// TIA Portal project "Snake" (V16)

(* hardware
DEVICE "S71500/ET200MP station_1"  S7-1500 station
   slot 0: "Telaio di montaggio_0"  Rack  6ES7 590-1***0-0AA0
   slot 1: "PLC_1"  CPU 1515-2 PN  6ES7 515-2AM02-0AB0  V2.8
      slot 3: "Display CPU_1"  6ES7591-1BA00-0AA0
      slot 32768: "Interfaccia PROFINET_1"  X1
         slot 32769: "Porta_1"  X1 P1
         slot 32770: "Porta_2"  X1 P2
      slot 33024: "Interfaccia PROFINET_2"  X2
         slot 33025: "Porta_1"  X2 P1
      slot 34817: "Virtual CP interface port_1"  Virtual CP interface port  Virtual CP interface port
DEVICE "HMI_1"  TP2200 Comfort
   slot 0: "HMI_1"  TP2200 Comfort  6AV2 124-0XC02-0AX1  16.0.0.0
   slot 1: "HMI_RT_2"  TP2200 Comfort  6AV2 124-0XC02-0AX1  16.0.0.0
   slot 5: "HMI_1.IE_CP_1"  PROFINET Interface  16.0.0.0
      slot 1: "Interfaccia_1 PROFINET"  PROFINET Interface
         slot 1: "Porta_1"  Port
         slot 2: "Porta_2"  Port
   slot 6: "HMI_1.IE_CP_2"  PROFINET Interface  16.0.0.0
      slot 1: "PROFINET Interface_GBit"  PROFINET Interface
         slot 1: "Porta_1"  Port
   slot 7: "HMI_1.MPI/DP_CP_1"  MPI/DP Interface  16.0.0.0
*)

// ===== PLC "PLC_1"  CPU 1515-2 PN =====

VAR_GLOBAL CONSTANT   // PLC tag table "Constants"
   "SNAKE_START_NUM" : DInt := 3;
   "DIRECTION_UP" : Int := 1;
   "DIRECTION_DOWN" : Int := 2;
   "DIRECTION_RIGHT" : Int := 3;
   "DIRECTION_LEFT" : Int := 4;
   "FIELD_HEIGHT" : DInt := 10;
   "FIELD_LENGTH" : DInt := 20;
   "DIRECTION_NONE" : Int := 0;
   "POINTS_BASE" : UDInt := 50;
END_VAR

TYPE "st_FieldBlock"
   STRUCT
      SnakePresence : Bool;   // Snake block present
      ApplePresence : Bool;   // Apple block present
      Shifted : Bool;   // Block already shifted
      PreviousDirection : Int;   // Previous block direction (1 = Up, 2 = Down, 3 = Right, 4 = Left)
      HMI_Visualization : USInt;   // HMI visualization (0 = nothing / 1 = snake / 2 = apple)
   END_STRUCT;
END_TYPE

DATA_BLOCK "DB_Field"   // DB1
{ S7_Optimized_Access := 'TRUE' }
VERSION : 0.1
   VAR RETAIN
      Field : Array[1.."FIELD_HEIGHT", 1.."FIELD_LENGTH"] of "st_FieldBlock";
   END_VAR
BEGIN
END_DATA_BLOCK

DATA_BLOCK "DB_Commands"   // DB2
{ S7_Optimized_Access := 'TRUE' }
VERSION : 0.1
   VAR
      Cmd : Struct
         Start : Bool;   // Start command
         Stop : Bool;   // Stop command
         Pause : Bool;   // Pause command
         SnakeUp : Bool;
         SnakeDown : Bool;
         SnakeRight : Bool;
         SnakeLeft : Bool;
         Speed : Real;   // Speed (blocks per second)
      END_STRUCT;
      Sts : Struct
         GameActive : Bool;   // Game active
         PauseActive : Bool;   // Pause active
         SnakeLength : UDInt;
      END_STRUCT;
   END_VAR
   VAR RETAIN
      Points : Struct
         Actual : UDInt;
         LastGame : UDInt;
         BestGame : UDInt;
         BestLength : UDInt;
      END_STRUCT;
   END_VAR
BEGIN
END_DATA_BLOCK

DATA_BLOCK "FB_MainLogic_DB"   // DB3
{ S7_Optimized_Access := 'TRUE' }
VERSION : 0.1
// stored: InstanceOfName FB_MainLogic
"FB_MainLogic"
BEGIN
END_DATA_BLOCK

FUNCTION_BLOCK "FB_MainLogic"   // FB1, SCL
{ S7_Optimized_Access := 'TRUE' }
VERSION : 0.1
   VAR
      TON_Speed : TON_TIME;   // Timer used for game speed
      ResetTimer : Bool;
      Fp_GameStart : R_TRIG;   // Edge detection for game start
      Fn_GameStart : F_TRIG;
      SnakeHeadHeightIndex : DInt;   // Height index for snake head (used for starting the calculation loops for the movement)
      SnakeHeadLengthIndex : DInt;   // Length index for snake head (used for starting the calculation loops for the movement)
      PreviousDirection : Int;
      SnakeDirection : Int;   // Snake Direction
   END_VAR
   VAR_TEMP
      PointsToAdd : UDInt;
      IndexHeight : DInt;
      IndexLength : DInt;
      RandomAppleHeight : DInt;   // Random height index where to generate the apple
      RandomAppleLength : DInt;   // Random length index where to generate the apple
      CollisionWithSnake : Bool;
      CollisionWithWall : Bool;
      GenerateApple : Bool;
      ShiftFlag : Bool;   // Variable for snake movement
      LengthIndexToCheck : DInt;
      HeightIndexToCheck : DInt;
      CheckSnakeLength : UDInt;
      DirectionToCheck : Int;
   END_VAR
BEGIN

   REGION Game commands

       REGION Game start

           IF "DB_Commands".Cmd.Start AND NOT "DB_Commands".Sts.GameActive THEN
               IF "DB_Commands".Cmd.Speed > 0.0 THEN
                   "DB_Commands".Sts.GameActive := TRUE;
                   "DB_Commands".Sts.PauseActive := FALSE;
               END_IF;
               "DB_Commands".Cmd.Start := FALSE;
           ELSIF "DB_Commands".Sts.GameActive THEN
               "DB_Commands".Cmd.Start := FALSE;
           END_IF;

       END_REGION

       REGION Game stop

           IF "DB_Commands".Cmd.Stop OR ("DB_Commands".Cmd.Speed <= 0.0) THEN
               "DB_Commands".Sts.GameActive := FALSE;
               "DB_Commands".Sts.PauseActive := FALSE;
               "DB_Commands".Cmd.Stop := FALSE;
               "DB_Commands".Cmd.Start := FALSE;
           END_IF;

       END_REGION

       REGION Game Pause

           IF "DB_Commands".Cmd.Pause THEN
               IF "DB_Commands".Sts.GameActive THEN
                   "DB_Commands".Sts.PauseActive := NOT "DB_Commands".Sts.PauseActive;
               ELSE
                   "DB_Commands".Sts.PauseActive := FALSE;
               END_IF;
               "DB_Commands".Cmd.Pause := FALSE;
           END_IF;

       END_REGION

       REGION Game speed

           IF "DB_Commands".Cmd.Speed > 0.0 THEN

               #TON_Speed(IN := "DB_Commands".Sts.GameActive AND NOT "DB_Commands".Sts.PauseActive AND NOT #ResetTimer,
                          PT := REAL_TO_DINT((1.0 / "DB_Commands".Cmd.Speed) * 1000.0));

               #ResetTimer := #TON_Speed.Q;
               #ShiftFlag := #TON_Speed.Q;

           END_IF;

       END_REGION

       REGION Game points

           #PointsToAdd := REAL_TO_UDINT("DB_Commands".Cmd.Speed * UDINT_TO_REAL("POINTS_BASE"));

       END_REGION

       REGION Snake movements

           IF "DB_Commands".Sts.GameActive AND NOT "DB_Commands".Sts.PauseActive THEN

               IF #ShiftFlag THEN

                   //Up
                   IF "DB_Commands".Cmd.SnakeUp THEN
                       IF #SnakeDirection <> "DIRECTION_DOWN" THEN
                           #SnakeDirection := "DIRECTION_UP";
                       END_IF;
                       "DB_Commands".Cmd.SnakeUp := FALSE;
                       //Down
                   ELSIF "DB_Commands".Cmd.SnakeDown THEN
                       IF #SnakeDirection <> "DIRECTION_UP" THEN
                           #SnakeDirection := "DIRECTION_DOWN";
                       END_IF;
                       "DB_Commands".Cmd.SnakeDown := FALSE;
                       //Left
                   ELSIF "DB_Commands".Cmd.SnakeLeft THEN
                       IF #SnakeDirection <> "DIRECTION_RIGHT" THEN
                           #SnakeDirection := "DIRECTION_LEFT";
                       END_IF;
                       "DB_Commands".Cmd.SnakeLeft := FALSE;
                       //Right
                   ELSIF "DB_Commands".Cmd.SnakeRight THEN
                       IF #SnakeDirection <> "DIRECTION_LEFT" THEN
                           #SnakeDirection := "DIRECTION_RIGHT";
                       END_IF;
                       "DB_Commands".Cmd.SnakeRight := FALSE;
                   END_IF;

               END_IF;

           ELSE
               "DB_Commands".Cmd.SnakeUp := FALSE;
               "DB_Commands".Cmd.SnakeDown := FALSE;
               "DB_Commands".Cmd.SnakeLeft := FALSE;
               "DB_Commands".Cmd.SnakeRight := FALSE;
           END_IF;

       END_REGION

   END_REGION


   REGION Game logic

       REGION Check start and snake + apple creation

           #Fp_GameStart(CLK := "DB_Commands".Sts.GameActive);

           IF #Fp_GameStart.Q THEN

               //Reset actual points
               "DB_Commands".Points.Actual := 0;

               //Reset previous game
               FOR #IndexHeight := 1 TO "FIELD_HEIGHT" DO
                   FOR #IndexLength := 1 TO "FIELD_LENGTH" DO
                       "DB_Field".Field[#IndexHeight, #IndexLength].SnakePresence := FALSE;
                       "DB_Field".Field[#IndexHeight, #IndexLength].ApplePresence := FALSE;
                       "DB_Field".Field[#IndexHeight, #IndexLength].PreviousDirection := "DIRECTION_NONE";
                       "DB_Field".Field[#IndexHeight, #IndexLength].Shifted := FALSE;
                   END_FOR;
               END_FOR;

               //Check for starting indexes
               #SnakeHeadHeightIndex := "FIELD_HEIGHT" / 2; //5
               #SnakeHeadLengthIndex := "FIELD_LENGTH" / 2; //10

               //Set right direction for starting
               #SnakeDirection := #PreviousDirection := "DIRECTION_RIGHT";

               FOR #IndexLength := #SnakeHeadLengthIndex TO (#SnakeHeadLengthIndex - "SNAKE_START_NUM" + 1) BY -1 DO
                   "DB_Field".Field[#SnakeHeadHeightIndex, #IndexLength].SnakePresence := TRUE;
                   "DB_Field".Field[#SnakeHeadHeightIndex, #IndexLength].PreviousDirection := #SnakeDirection;
                   //Check for index bound
                   IF #IndexLength <= 1 THEN
                       EXIT;
                   END_IF;
               END_FOR;

               REGION Random number generation for apple

                   //Generate random number for apple creation
                   #RandomAppleHeight := "FC_RandomGen"(LowerLimit := 1, UpperLimit := "FIELD_HEIGHT");
                   #RandomAppleLength := "FC_RandomGen"(LowerLimit := 1, UpperLimit := "FIELD_LENGTH");

                   //Check if the numbers set are not already a snake block
                   WHILE "DB_Field".Field[#RandomAppleHeight, #RandomAppleLength].SnakePresence DO
                       //First time checking
                       IF NOT "DB_Field".Field[#RandomAppleHeight, #RandomAppleLength].SnakePresence THEN
                           EXIT;
                       END_IF;

                       //If there's the snake then change indexes
                       #RandomAppleHeight := #RandomAppleHeight + "FC_RandomGen"(LowerLimit := 1, UpperLimit := "FIELD_HEIGHT");
                       #RandomAppleHeight := #RandomAppleHeight MOD "FIELD_HEIGHT";
                       #RandomAppleLength := #RandomAppleLength + "FC_RandomGen"(LowerLimit := 1, UpperLimit := "FIELD_LENGTH");
                       #RandomAppleLength := #RandomAppleLength MOD "FIELD_LENGTH";

                   END_WHILE;

                   //Set apple presence
                   "DB_Field".Field[#RandomAppleHeight, #RandomAppleLength].ApplePresence := TRUE;

               END_REGION

           END_IF;

       END_REGION

       REGION Snake movement

           IF #ShiftFlag THEN

               //Reset collisions & vars
               #CollisionWithSnake := FALSE;
               #CollisionWithWall := FALSE;
               #GenerateApple := FALSE;

               //Reset Shifted vars
               FOR #IndexHeight := 1 TO "FIELD_HEIGHT" DO
                   FOR #IndexLength := 1 TO "FIELD_LENGTH" DO
                       "DB_Field".Field[#IndexHeight, #IndexLength].Shifted := FALSE;
                   END_FOR;
               END_FOR;

               //Check snake movement
               IF #SnakeDirection = "DIRECTION_RIGHT" THEN

                   REGION Right direction

                       //Check wall collision
                       IF (#SnakeHeadLengthIndex + 1) > "FIELD_LENGTH" THEN
                           #CollisionWithWall := TRUE;
                           "DB_Commands".Sts.GameActive := FALSE;
                       ELSE
                           //Check collision with other snake parts
                           IF "DB_Field".Field[#SnakeHeadHeightIndex, #SnakeHeadLengthIndex + 1].SnakePresence THEN
                               #CollisionWithSnake := TRUE;
                               "DB_Commands".Sts.GameActive := FALSE;
                           END_IF;
                       END_IF;

                       //Move if we have no collisions
                       IF NOT #CollisionWithWall AND NOT #CollisionWithSnake THEN
                           //Right direction starting with the head
                           //Shift snake head
                           "DB_Field".Field[#SnakeHeadHeightIndex, #SnakeHeadLengthIndex + 1].SnakePresence := "DB_Field".Field[#SnakeHeadHeightIndex, #SnakeHeadLengthIndex].SnakePresence;
                           "DB_Field".Field[#SnakeHeadHeightIndex, #SnakeHeadLengthIndex + 1].Shifted := TRUE;
                           "DB_Field".Field[#SnakeHeadHeightIndex, #SnakeHeadLengthIndex + 1].PreviousDirection := #PreviousDirection := "DIRECTION_RIGHT";
                           //If apple presence in the block then don't delete the snake presence to create the new block
                           IF "DB_Field".Field[#SnakeHeadHeightIndex, #SnakeHeadLengthIndex + 1].ApplePresence THEN
                               "DB_Field".Field[#SnakeHeadHeightIndex, #SnakeHeadLengthIndex + 1].ApplePresence := FALSE;
                               "DB_Field".Field[#SnakeHeadHeightIndex, #SnakeHeadLengthIndex].Shifted := TRUE;
                               "DB_Field".Field[#SnakeHeadHeightIndex, #SnakeHeadLengthIndex].PreviousDirection := "DIRECTION_RIGHT";
                               #GenerateApple := TRUE;
                           ELSE
                               "DB_Field".Field[#SnakeHeadHeightIndex, #SnakeHeadLengthIndex].SnakePresence := FALSE;
                               "DB_Field".Field[#SnakeHeadHeightIndex, #SnakeHeadLengthIndex].PreviousDirection := "DIRECTION_NONE";
                           END_IF;
                           //Set the new direction to check for snake movement
                           #DirectionToCheck := "DIRECTION_LEFT";
                           #LengthIndexToCheck := #SnakeHeadLengthIndex;
                           #HeightIndexToCheck := #SnakeHeadHeightIndex;
                           //And update the new snake head indexes
                           #SnakeHeadLengthIndex := #SnakeHeadLengthIndex + 1;

                       END_IF;

                   END_REGION

               ELSIF #SnakeDirection = "DIRECTION_LEFT" THEN

                   REGION Left direction

                       //Check wall collision
                       IF (#SnakeHeadLengthIndex - 1) < 1 THEN
                           #CollisionWithWall := TRUE;
                           "DB_Commands".Sts.GameActive := FALSE;
                       ELSE
                           //Check collision with other snake parts
                           IF "DB_Field".Field[#SnakeHeadHeightIndex, #SnakeHeadLengthIndex - 1].SnakePresence THEN
                               #CollisionWithSnake := TRUE;
                               "DB_Commands".Sts.GameActive := FALSE;
                           END_IF;
                       END_IF;

                       //Move if we have no collisions
                       IF NOT #CollisionWithWall AND NOT #CollisionWithSnake THEN
                           //Right direction starting with the head
                           //Shift snake head
                           "DB_Field".Field[#SnakeHeadHeightIndex, #SnakeHeadLengthIndex - 1].SnakePresence := "DB_Field".Field[#SnakeHeadHeightIndex, #SnakeHeadLengthIndex].SnakePresence;
                           "DB_Field".Field[#SnakeHeadHeightIndex, #SnakeHeadLengthIndex - 1].Shifted := TRUE;
                           "DB_Field".Field[#SnakeHeadHeightIndex, #SnakeHeadLengthIndex - 1].PreviousDirection := #PreviousDirection := "DIRECTION_LEFT";
                           //If apple presence in the block then don't delete the snake presence to create the new block
                           IF "DB_Field".Field[#SnakeHeadHeightIndex, #SnakeHeadLengthIndex - 1].ApplePresence THEN
                               "DB_Field".Field[#SnakeHeadHeightIndex, #SnakeHeadLengthIndex - 1].ApplePresence := FALSE;
                               "DB_Field".Field[#SnakeHeadHeightIndex, #SnakeHeadLengthIndex].Shifted := TRUE;
                               "DB_Field".Field[#SnakeHeadHeightIndex, #SnakeHeadLengthIndex].PreviousDirection := "DIRECTION_LEFT";
                               #GenerateApple := TRUE;
                           ELSE
                               "DB_Field".Field[#SnakeHeadHeightIndex, #SnakeHeadLengthIndex].SnakePresence := FALSE;
                               "DB_Field".Field[#SnakeHeadHeightIndex, #SnakeHeadLengthIndex].PreviousDirection := "DIRECTION_NONE";
                           END_IF;
                           //Set the new direction to check for snake movement
                           #DirectionToCheck := "DIRECTION_RIGHT";
                           #LengthIndexToCheck := #SnakeHeadLengthIndex;
                           #HeightIndexToCheck := #SnakeHeadHeightIndex;
                           //And update the new snake head indexes
                           #SnakeHeadLengthIndex := #SnakeHeadLengthIndex - 1;

                       END_IF;

                   END_REGION

               ELSIF #SnakeDirection = "DIRECTION_UP" THEN

                   REGION Up direction

                       //Check wall collision
                       IF (#SnakeHeadHeightIndex + 1) > "FIELD_HEIGHT" THEN
                           #CollisionWithWall := TRUE;
                           "DB_Commands".Sts.GameActive := FALSE;
                       ELSE
                           //Check collision with other snake parts
                           IF "DB_Field".Field[#SnakeHeadHeightIndex + 1, #SnakeHeadLengthIndex].SnakePresence THEN
                               #CollisionWithSnake := TRUE;
                               "DB_Commands".Sts.GameActive := FALSE;
                           END_IF;
                       END_IF;

                       //Move if we have no collisions
                       IF NOT #CollisionWithWall AND NOT #CollisionWithSnake THEN
                           //Right direction starting with the head
                           //Shift snake head
                           "DB_Field".Field[#SnakeHeadHeightIndex + 1, #SnakeHeadLengthIndex].SnakePresence := "DB_Field".Field[#SnakeHeadHeightIndex, #SnakeHeadLengthIndex].SnakePresence;
                           "DB_Field".Field[#SnakeHeadHeightIndex + 1, #SnakeHeadLengthIndex].Shifted := TRUE;
                           "DB_Field".Field[#SnakeHeadHeightIndex + 1, #SnakeHeadLengthIndex].PreviousDirection := #PreviousDirection := "DIRECTION_UP";
                           //If apple presence in the block then don't delete the snake presence to create the new block
                           IF "DB_Field".Field[#SnakeHeadHeightIndex + 1, #SnakeHeadLengthIndex].ApplePresence THEN
                               "DB_Field".Field[#SnakeHeadHeightIndex + 1, #SnakeHeadLengthIndex].ApplePresence := FALSE;
                               "DB_Field".Field[#SnakeHeadHeightIndex, #SnakeHeadLengthIndex].Shifted := TRUE;
                               "DB_Field".Field[#SnakeHeadHeightIndex, #SnakeHeadLengthIndex].PreviousDirection := "DIRECTION_UP";
                               #GenerateApple := TRUE;
                           ELSE
                               "DB_Field".Field[#SnakeHeadHeightIndex, #SnakeHeadLengthIndex].SnakePresence := FALSE;
                               "DB_Field".Field[#SnakeHeadHeightIndex, #SnakeHeadLengthIndex].PreviousDirection := "DIRECTION_NONE";
                           END_IF;
                           //Set the new direction to check for snake movement
                           #DirectionToCheck := "DIRECTION_DOWN";
                           #LengthIndexToCheck := #SnakeHeadLengthIndex;
                           #HeightIndexToCheck := #SnakeHeadHeightIndex;
                           //And update the new snake head indexes
                           #SnakeHeadHeightIndex := #SnakeHeadHeightIndex + 1;

                       END_IF;

                   END_REGION

               ELSIF #SnakeDirection = "DIRECTION_DOWN" THEN

                   REGION Down direction

                       //Check wall collision
                       IF (#SnakeHeadHeightIndex - 1) < 1 THEN
                           #CollisionWithWall := TRUE;
                           "DB_Commands".Sts.GameActive := FALSE;
                       ELSE
                           //Check collision with other snake parts
                           IF "DB_Field".Field[#SnakeHeadHeightIndex - 1, #SnakeHeadLengthIndex].SnakePresence THEN
                               #CollisionWithSnake := TRUE;
                               "DB_Commands".Sts.GameActive := FALSE;
                           END_IF;
                       END_IF;

                       //Move if we have no collisions
                       IF NOT #CollisionWithWall AND NOT #CollisionWithSnake THEN
                           //Right direction starting with the head
                           //Shift snake head
                           "DB_Field".Field[#SnakeHeadHeightIndex - 1, #SnakeHeadLengthIndex].SnakePresence := "DB_Field".Field[#SnakeHeadHeightIndex, #SnakeHeadLengthIndex].SnakePresence;
                           "DB_Field".Field[#SnakeHeadHeightIndex - 1, #SnakeHeadLengthIndex].Shifted := TRUE;
                           "DB_Field".Field[#SnakeHeadHeightIndex - 1, #SnakeHeadLengthIndex].PreviousDirection := #PreviousDirection := "DIRECTION_DOWN";
                           //If apple presence in the block then don't delete the snake presence to create the new block
                           IF "DB_Field".Field[#SnakeHeadHeightIndex - 1, #SnakeHeadLengthIndex].ApplePresence THEN
                               "DB_Field".Field[#SnakeHeadHeightIndex - 1, #SnakeHeadLengthIndex].ApplePresence := FALSE;
                               "DB_Field".Field[#SnakeHeadHeightIndex, #SnakeHeadLengthIndex].Shifted := TRUE;
                               "DB_Field".Field[#SnakeHeadHeightIndex, #SnakeHeadLengthIndex].PreviousDirection := "DIRECTION_DOWN";
                               #GenerateApple := TRUE;
                           ELSE
                               "DB_Field".Field[#SnakeHeadHeightIndex, #SnakeHeadLengthIndex].SnakePresence := FALSE;
                               "DB_Field".Field[#SnakeHeadHeightIndex, #SnakeHeadLengthIndex].PreviousDirection := "DIRECTION_NONE";
                           END_IF;
                           //Set the new direction to check for snake movement
                           #DirectionToCheck := "DIRECTION_UP";
                           #LengthIndexToCheck := #SnakeHeadLengthIndex;
                           #HeightIndexToCheck := #SnakeHeadHeightIndex;
                           //And update the new snake head indexes
                           #SnakeHeadHeightIndex := #SnakeHeadHeightIndex - 1;

                       END_IF;

                   END_REGION

               END_IF;

               REGION Snake shifts

                   IF NOT #CollisionWithWall AND NOT #CollisionWithSnake AND NOT #GenerateApple THEN

                       WHILE #DirectionToCheck <> "DIRECTION_NONE" DO

                           //Check the left direction
                           IF #DirectionToCheck = "DIRECTION_LEFT" THEN
                               FOR #IndexLength := (#LengthIndexToCheck - 1) TO 1 BY -1 DO
                                   IF "DB_Field".Field[#HeightIndexToCheck, #IndexLength].SnakePresence AND
                                       NOT "DB_Field".Field[#HeightIndexToCheck, #IndexLength].Shifted AND
                                       "DB_Field".Field[#HeightIndexToCheck, #IndexLength].PreviousDirection <> "DIRECTION_LEFT" THEN

                                       "DB_Field".Field[#HeightIndexToCheck, #IndexLength + 1].SnakePresence := "DB_Field".Field[#HeightIndexToCheck, #IndexLength].SnakePresence;
                                       "DB_Field".Field[#HeightIndexToCheck, #IndexLength + 1].PreviousDirection := #PreviousDirection;
                                       "DB_Field".Field[#HeightIndexToCheck, #IndexLength + 1].Shifted := TRUE;

                                       "DB_Field".Field[#HeightIndexToCheck, #IndexLength].SnakePresence := FALSE;
                                       "DB_Field".Field[#HeightIndexToCheck, #IndexLength].PreviousDirection := "DIRECTION_NONE";
                                       #LengthIndexToCheck := #IndexLength;
                                   ELSE
                                       EXIT;
                                   END_IF;
                               END_FOR;
                               //When the shift is finished check the other directions
                               #DirectionToCheck := "DIRECTION_NONE";
                               //Check up
                               IF (#HeightIndexToCheck + 1) <= "FIELD_HEIGHT" THEN
                                   IF "DB_Field".Field[#HeightIndexToCheck + 1, #LengthIndexToCheck].SnakePresence AND
                                       NOT "DB_Field".Field[#HeightIndexToCheck + 1, #LengthIndexToCheck].Shifted THEN
                                       #DirectionToCheck := "DIRECTION_UP";
                                       #PreviousDirection := "DIRECTION_DOWN";
                                   END_IF;
                               END_IF;
                               //Check down
                               IF (#HeightIndexToCheck - 1) >= 1 THEN
                                   IF "DB_Field".Field[#HeightIndexToCheck - 1, #LengthIndexToCheck].SnakePresence AND
                                       NOT "DB_Field".Field[#HeightIndexToCheck - 1, #LengthIndexToCheck].Shifted THEN
                                       #DirectionToCheck := "DIRECTION_DOWN";
                                       #PreviousDirection := "DIRECTION_UP";
                                   END_IF;
                               END_IF;

                               //Check the right direction
                           ELSIF #DirectionToCheck = "DIRECTION_RIGHT" THEN
                               FOR #IndexLength := (#LengthIndexToCheck + 1) TO "FIELD_LENGTH" DO
                                   IF "DB_Field".Field[#HeightIndexToCheck, #IndexLength].SnakePresence AND
                                       NOT "DB_Field".Field[#HeightIndexToCheck, #IndexLength].Shifted AND
                                       "DB_Field".Field[#HeightIndexToCheck, #IndexLength].PreviousDirection <> "DIRECTION_RIGHT" THEN

                                       "DB_Field".Field[#HeightIndexToCheck, #IndexLength - 1].SnakePresence := "DB_Field".Field[#HeightIndexToCheck, #IndexLength].SnakePresence;
                                       "DB_Field".Field[#HeightIndexToCheck, #IndexLength - 1].PreviousDirection := #PreviousDirection;
                                       "DB_Field".Field[#HeightIndexToCheck, #IndexLength - 1].Shifted := TRUE;

                                       "DB_Field".Field[#HeightIndexToCheck, #IndexLength].SnakePresence := FALSE;
                                       "DB_Field".Field[#HeightIndexToCheck, #IndexLength].PreviousDirection := "DIRECTION_NONE";
                                       #LengthIndexToCheck := #IndexLength;
                                   ELSE
                                       EXIT;
                                   END_IF;
                               END_FOR;
                               //When the shift is finished check the other directions
                               #DirectionToCheck := "DIRECTION_NONE";
                               //Check up
                               IF (#HeightIndexToCheck + 1) <= "FIELD_HEIGHT" THEN
                                   IF "DB_Field".Field[#HeightIndexToCheck + 1, #LengthIndexToCheck].SnakePresence AND
                                       NOT "DB_Field".Field[#HeightIndexToCheck + 1, #LengthIndexToCheck].Shifted THEN
                                       #DirectionToCheck := "DIRECTION_UP";
                                       #PreviousDirection := "DIRECTION_DOWN";
                                   END_IF;
                               END_IF;
                               //Check down
                               IF (#HeightIndexToCheck - 1) >= 1 THEN
                                   IF "DB_Field".Field[#HeightIndexToCheck - 1, #LengthIndexToCheck].SnakePresence AND
                                       NOT "DB_Field".Field[#HeightIndexToCheck - 1, #LengthIndexToCheck].Shifted THEN
                                       #DirectionToCheck := "DIRECTION_DOWN";
                                       #PreviousDirection := "DIRECTION_UP";
                                   END_IF;
                               END_IF;

                               //Check the down direction
                           ELSIF #DirectionToCheck = "DIRECTION_DOWN" THEN
                               FOR #IndexHeight := (#HeightIndexToCheck - 1) TO 1 BY -1 DO
                                   IF "DB_Field".Field[#IndexHeight, #LengthIndexToCheck].SnakePresence AND
                                       NOT "DB_Field".Field[#IndexHeight, #LengthIndexToCheck].Shifted AND
                                       "DB_Field".Field[#IndexHeight, #LengthIndexToCheck].PreviousDirection <> "DIRECTION_DOWN" THEN

                                       "DB_Field".Field[#IndexHeight + 1, #LengthIndexToCheck].SnakePresence := "DB_Field".Field[#IndexHeight, #LengthIndexToCheck].SnakePresence;
                                       "DB_Field".Field[#IndexHeight + 1, #LengthIndexToCheck].PreviousDirection := #PreviousDirection;
                                       "DB_Field".Field[#IndexHeight + 1, #LengthIndexToCheck].Shifted := TRUE;

                                       "DB_Field".Field[#IndexHeight, #LengthIndexToCheck].SnakePresence := FALSE;
                                       "DB_Field".Field[#IndexHeight, #LengthIndexToCheck].PreviousDirection := "DIRECTION_NONE";
                                       #HeightIndexToCheck := #IndexHeight;
                                   ELSE
                                       EXIT;
                                   END_IF;
                               END_FOR;
                               //When the shift is finished check the other directions
                               #DirectionToCheck := "DIRECTION_NONE";
                               //Check left
                               IF (#LengthIndexToCheck - 1) >= 1 THEN
                                   IF "DB_Field".Field[#HeightIndexToCheck, #LengthIndexToCheck - 1].SnakePresence AND
                                       NOT "DB_Field".Field[#HeightIndexToCheck, #LengthIndexToCheck - 1].Shifted THEN
                                       #DirectionToCheck := "DIRECTION_LEFT";
                                       #PreviousDirection := "DIRECTION_RIGHT";
                                   END_IF;
                               END_IF;
                               //Check down
                               IF (#LengthIndexToCheck + 1) <= "FIELD_LENGTH" THEN
                                   IF "DB_Field".Field[#HeightIndexToCheck, #LengthIndexToCheck + 1].SnakePresence AND
                                       NOT "DB_Field".Field[#HeightIndexToCheck, #LengthIndexToCheck + 1].Shifted THEN
                                       #DirectionToCheck := "DIRECTION_RIGHT";
                                       #PreviousDirection := "DIRECTION_LEFT";
                                   END_IF;
                               END_IF;

                               //Check the up direction
                           ELSIF #DirectionToCheck = "DIRECTION_UP" THEN
                               FOR #IndexHeight := (#HeightIndexToCheck + 1) TO "FIELD_HEIGHT" DO
                                   IF "DB_Field".Field[#IndexHeight, #LengthIndexToCheck].SnakePresence AND
                                       NOT "DB_Field".Field[#IndexHeight, #LengthIndexToCheck].Shifted AND
                                       "DB_Field".Field[#IndexHeight, #LengthIndexToCheck].PreviousDirection <> "DIRECTION_UP" THEN

                                       "DB_Field".Field[#IndexHeight - 1, #LengthIndexToCheck].SnakePresence := "DB_Field".Field[#IndexHeight, #LengthIndexToCheck].SnakePresence;
                                       "DB_Field".Field[#IndexHeight - 1, #LengthIndexToCheck].PreviousDirection := #PreviousDirection;
                                       "DB_Field".Field[#IndexHeight - 1, #LengthIndexToCheck].Shifted := TRUE;

                                       "DB_Field".Field[#IndexHeight, #LengthIndexToCheck].SnakePresence := FALSE;
                                       "DB_Field".Field[#IndexHeight, #LengthIndexToCheck].PreviousDirection := "DIRECTION_NONE";
                                       #HeightIndexToCheck := #IndexHeight;
                                   ELSE
                                       EXIT;
                                   END_IF;
                               END_FOR;
                               //When the shift is finished check the other directions
                               #DirectionToCheck := "DIRECTION_NONE";
                               //Check left
                               IF (#LengthIndexToCheck - 1) >= 1 THEN
                                   IF "DB_Field".Field[#HeightIndexToCheck, #LengthIndexToCheck - 1].SnakePresence AND
                                       NOT "DB_Field".Field[#HeightIndexToCheck, #LengthIndexToCheck - 1].Shifted THEN
                                       #DirectionToCheck := "DIRECTION_LEFT";
                                       #PreviousDirection := "DIRECTION_RIGHT";
                                   END_IF;
                               END_IF;
                               //Check down
                               IF (#LengthIndexToCheck + 1) <= "FIELD_LENGTH" THEN
                                   IF "DB_Field".Field[#HeightIndexToCheck, #LengthIndexToCheck + 1].SnakePresence AND
                                       NOT "DB_Field".Field[#HeightIndexToCheck, #LengthIndexToCheck + 1].Shifted THEN
                                       #DirectionToCheck := "DIRECTION_RIGHT";
                                       #PreviousDirection := "DIRECTION_LEFT";
                                   END_IF;
                               END_IF;
                           END_IF;

                       END_WHILE;

                   END_IF;

               END_REGION

               REGION Check for new apple generation

                   IF #GenerateApple THEN

                       //Increase score
                       "DB_Commands".Points.Actual := "DB_Commands".Points.Actual + #PointsToAdd;

                       //Generate random number for apple creation
                       #RandomAppleHeight := "FC_RandomGen"(LowerLimit := 1, UpperLimit := "FIELD_HEIGHT");
                       #RandomAppleLength := "FC_RandomGen"(LowerLimit := 1, UpperLimit := "FIELD_LENGTH");

                       //Check if the numbers set are not already a snake block
                       WHILE "DB_Field".Field[#RandomAppleHeight, #RandomAppleLength].SnakePresence DO
                           //First time checking
                           IF NOT "DB_Field".Field[#RandomAppleHeight, #RandomAppleLength].SnakePresence THEN
                               EXIT;
                           END_IF;

                           //If there's the snake then change indexes
                           #RandomAppleHeight := #RandomAppleHeight + "FC_RandomGen"(LowerLimit := 1, UpperLimit := "FIELD_HEIGHT");
                           #RandomAppleHeight := #RandomAppleHeight MOD "FIELD_HEIGHT";
                           #RandomAppleLength := #RandomAppleLength + "FC_RandomGen"(LowerLimit := 1, UpperLimit := "FIELD_LENGTH");
                           #RandomAppleLength := #RandomAppleLength MOD "FIELD_LENGTH";

                       END_WHILE;

                       //Set apple presence
                       "DB_Field".Field[#RandomAppleHeight, #RandomAppleLength].ApplePresence := TRUE;

                   END_IF;

               END_REGION

           END_IF;

       END_REGION

       REGION Snake length calculation

           "DB_Commands".Sts.SnakeLength := 0;
           FOR #IndexHeight := 1 TO "FIELD_HEIGHT" DO
               FOR #IndexLength := 1 TO "FIELD_LENGTH" DO
                   IF "DB_Field".Field[#IndexHeight, #IndexLength].SnakePresence THEN
                       "DB_Commands".Sts.SnakeLength := "DB_Commands".Sts.SnakeLength + 1;
                   END_IF;
               END_FOR;
           END_FOR;

       END_REGION

       REGION Check for game end to score points

           #Fn_GameStart(CLK := "DB_Commands".Sts.GameActive);

           IF #Fn_GameStart.Q THEN
               "DB_Commands".Points.LastGame := "DB_Commands".Points.Actual;
               IF "DB_Commands".Points.LastGame > "DB_Commands".Points.BestGame THEN
                   "DB_Commands".Points.BestGame := "DB_Commands".Points.LastGame;
               END_IF;
               IF "DB_Commands".Sts.SnakeLength > "DB_Commands".Points.BestLength THEN
                   "DB_Commands".Points.BestLength := "DB_Commands".Sts.SnakeLength;
               END_IF;
           END_IF;

       END_REGION

   END_REGION
END_FUNCTION_BLOCK

FUNCTION "FC_RandomGen" : DInt   // FC1, LAD
{ S7_Optimized_Access := 'TRUE' }
VERSION : 0.1
   VAR_INPUT
      LowerLimit : DInt;
      UpperLimit : DInt;
   END_VAR
   VAR_TEMP
      DateTime : DTL;
      ReadTimeRetVal : Int;
      NanoSecMod : Int;
      ChoppedTime : Int;
      UShift : UInt;
      SemiRandom : UInt;
      NormalizedRandom : Real;
   END_VAR
BEGIN

REGION Network 1: Read actual date/time to retrieve nanoseconds
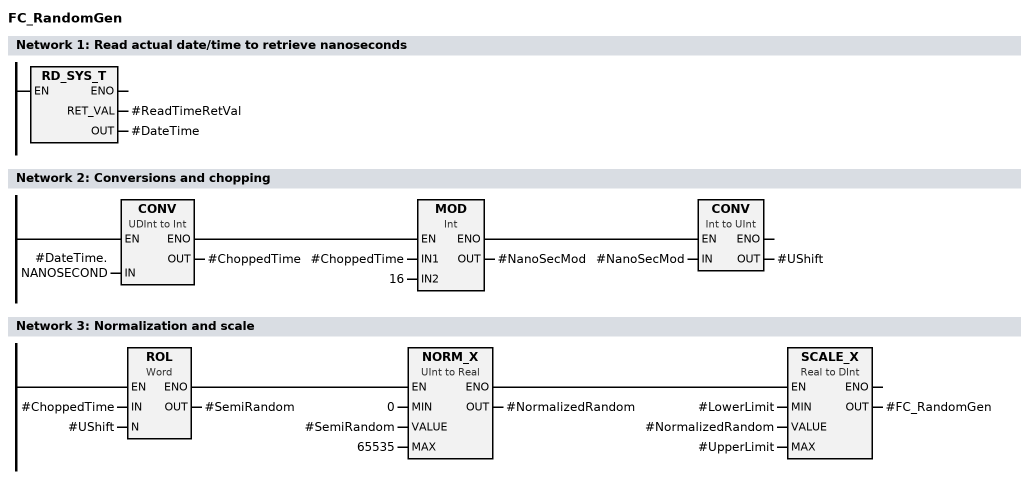
   #ReadTimeRetVal := RD_SYS_T(OUT => #DateTime);
END_REGION

REGION Network 2: Conversions and chopping
   RUNG wire#powerrail
      { S7_Templates := "[SrcType := UDInt, DestType := Int]" } Convert(in := #DateTime.NANOSECOND, out => #ChoppedTime)
      { S7_Templates := "SrcType := Int" } Mod(in1 := #ChoppedTime, in2 := 16, out => #NanoSecMod)
      { S7_Templates := "[SrcType := Int, DestType := UInt]" } Convert(in := #NanoSecMod, out => #UShift)
   END_RUNG
   // the same network as SCL:
   #ChoppedTime := UDINT_TO_INT(#DateTime.NANOSECOND);
   #NanoSecMod := #ChoppedTime MOD 16;
   #UShift := INT_TO_UINT(#NanoSecMod);
END_REGION

REGION Network 3: Normalization and scale
   #SemiRandom := ROL(IN := #ChoppedTime, N := #UShift);
   #NormalizedRandom := NORM_X(MIN := 0, VALUE := #SemiRandom, MAX := 65535);
   #FC_RandomGen := SCALE_X(MIN := #LowerLimit, VALUE := #NormalizedRandom, MAX := #UpperLimit);
END_REGION
END_FUNCTION

ORGANIZATION_BLOCK "Main"   // OB1, LAD, ProgramCycle
TITLE = "Main Program Sweep (Cycle)"
{ S7_Optimized_Access := 'TRUE' }
VERSION : 0.1
   VAR_INPUT
      Initial_Call : Bool;   // Initial call of this OB
      Remanence : Bool;   // =True, if remanent data are available
   END_VAR
   VAR_TEMP
      IndexHeight : DInt;
      IndexLength : DInt;
   END_VAR
BEGIN

REGION Network 1
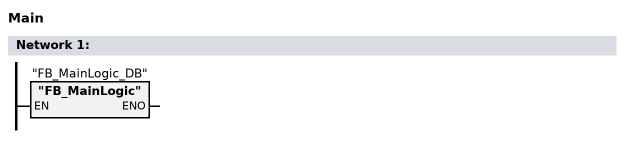
   RUNG wire#powerrail
      "FB_MainLogic_DB"()
   END_RUNG
   // the same network as SCL:
   "FB_MainLogic_DB"();   // "FB_MainLogic"
END_REGION

REGION Network 2 (SCL): Visualizzazione blocchi per HMI
   FOR #IndexHeight := 1 TO "FIELD_HEIGHT" DO
       FOR #IndexLength := 1 TO "FIELD_LENGTH" DO
           IF "DB_Field".Field[#IndexHeight, #IndexLength].SnakePresence THEN
               "DB_Field".Field[#IndexHeight, #IndexLength].HMI_Visualization := 1;
           ELSIF "DB_Field".Field[#IndexHeight, #IndexLength].ApplePresence THEN
               "DB_Field".Field[#IndexHeight, #IndexLength].HMI_Visualization := 2;
           ELSE
               "DB_Field".Field[#IndexHeight, #IndexLength].HMI_Visualization := 0;
           END_IF;
       END_FOR;
   END_FOR;
END_REGION
END_ORGANIZATION_BLOCK

(* ===== HMI "HMI_RT_2" =====
system functions are stored by id; their names below are inferred from use
connection "HMI_Collegamento_1": ETHERNET, S7_1500_OMS

HMI tags "Tabella delle variabili standard"
   "Variabile_Numero di pagina" : UInt, internal
   "DB_Field_Field{1,1}_HMI_Visualization" : USInt = PLC DB_Field.Field[1,1].HMI_Visualization AT %DB1.DBW0, 100 ms
   "DB_Field_Field{1,2}_HMI_Visualization" : USInt = PLC DB_Field.Field[1,2].HMI_Visualization AT %DB1.DBW0, 100 ms
   "DB_Field_Field{1,3}_HMI_Visualization" : USInt = PLC DB_Field.Field[1,3].HMI_Visualization AT %DB1.DBW0, 100 ms
   "DB_Field_Field{1,4}_HMI_Visualization" : USInt = PLC DB_Field.Field[1,4].HMI_Visualization AT %DB1.DBW0, 100 ms
   "DB_Field_Field{1,5}_HMI_Visualization" : USInt = PLC DB_Field.Field[1,5].HMI_Visualization AT %DB1.DBW0, 100 ms
   "DB_Field_Field{1,6}_HMI_Visualization" : USInt = PLC DB_Field.Field[1,6].HMI_Visualization AT %DB1.DBW0, 100 ms
   "DB_Field_Field{1,7}_HMI_Visualization" : USInt = PLC DB_Field.Field[1,7].HMI_Visualization AT %DB1.DBW0, 100 ms
   "DB_Field_Field{1,8}_HMI_Visualization" : USInt = PLC DB_Field.Field[1,8].HMI_Visualization AT %DB1.DBW0, 100 ms
   "DB_Field_Field{1,9}_HMI_Visualization" : USInt = PLC DB_Field.Field[1,9].HMI_Visualization AT %DB1.DBW0, 100 ms
   "DB_Field_Field{1,10}_HMI_Visualization" : USInt = PLC DB_Field.Field[1,10].HMI_Visualization AT %DB1.DBW0, 100 ms
   "DB_Field_Field{1,11}_HMI_Visualization" : USInt = PLC DB_Field.Field[1,11].HMI_Visualization AT %DB1.DBW0, 100 ms
   "DB_Field_Field{1,12}_HMI_Visualization" : USInt = PLC DB_Field.Field[1,12].HMI_Visualization AT %DB1.DBW0, 100 ms
   "DB_Field_Field{1,13}_HMI_Visualization" : USInt = PLC DB_Field.Field[1,13].HMI_Visualization AT %DB1.DBW0, 100 ms
   "DB_Field_Field{1,14}_HMI_Visualization" : USInt = PLC DB_Field.Field[1,14].HMI_Visualization AT %DB1.DBW0, 100 ms
   "DB_Field_Field{1,15}_HMI_Visualization" : USInt = PLC DB_Field.Field[1,15].HMI_Visualization AT %DB1.DBW0, 100 ms
   "DB_Field_Field{1,16}_HMI_Visualization" : USInt = PLC DB_Field.Field[1,16].HMI_Visualization AT %DB1.DBW0, 100 ms
   "DB_Field_Field{1,17}_HMI_Visualization" : USInt = PLC DB_Field.Field[1,17].HMI_Visualization AT %DB1.DBW0, 100 ms
   "DB_Field_Field{1,18}_HMI_Visualization" : USInt = PLC DB_Field.Field[1,18].HMI_Visualization AT %DB1.DBW0, 100 ms
   "DB_Field_Field{1,19}_HMI_Visualization" : USInt = PLC DB_Field.Field[1,19].HMI_Visualization AT %DB1.DBW0, 100 ms
   "DB_Field_Field{1,20}_HMI_Visualization" : USInt = PLC DB_Field.Field[1,20].HMI_Visualization AT %DB1.DBW0, 100 ms
   "DB_Field_Field{2,1}_HMI_Visualization" : USInt = PLC DB_Field.Field[2,1].HMI_Visualization AT %DB1.DBW0, 100 ms
   "DB_Field_Field{2,2}_HMI_Visualization" : USInt = PLC DB_Field.Field[2,2].HMI_Visualization AT %DB1.DBW0, 100 ms
   "DB_Field_Field{2,3}_HMI_Visualization" : USInt = PLC DB_Field.Field[2,3].HMI_Visualization AT %DB1.DBW0, 100 ms
   "DB_Field_Field{2,4}_HMI_Visualization" : USInt = PLC DB_Field.Field[2,4].HMI_Visualization AT %DB1.DBW0, 100 ms
   "DB_Field_Field{2,5}_HMI_Visualization" : USInt = PLC DB_Field.Field[2,5].HMI_Visualization AT %DB1.DBW0, 100 ms
   "DB_Field_Field{2,6}_HMI_Visualization" : USInt = PLC DB_Field.Field[2,6].HMI_Visualization AT %DB1.DBW0, 100 ms
   "DB_Field_Field{2,7}_HMI_Visualization" : USInt = PLC DB_Field.Field[2,7].HMI_Visualization AT %DB1.DBW0, 100 ms
   "DB_Field_Field{2,8}_HMI_Visualization" : USInt = PLC DB_Field.Field[2,8].HMI_Visualization AT %DB1.DBW0, 100 ms
   "DB_Field_Field{2,9}_HMI_Visualization" : USInt = PLC DB_Field.Field[2,9].HMI_Visualization AT %DB1.DBW0, 100 ms
   "DB_Field_Field{2,10}_HMI_Visualization" : USInt = PLC DB_Field.Field[2,10].HMI_Visualization AT %DB1.DBW0, 100 ms
   "DB_Field_Field{2,11}_HMI_Visualization" : USInt = PLC DB_Field.Field[2,11].HMI_Visualization AT %DB1.DBW0, 100 ms
   "DB_Field_Field{2,12}_HMI_Visualization" : USInt = PLC DB_Field.Field[2,12].HMI_Visualization AT %DB1.DBW0, 100 ms
   "DB_Field_Field{2,13}_HMI_Visualization" : USInt = PLC DB_Field.Field[2,13].HMI_Visualization AT %DB1.DBW0, 100 ms
   "DB_Field_Field{2,14}_HMI_Visualization" : USInt = PLC DB_Field.Field[2,14].HMI_Visualization AT %DB1.DBW0, 100 ms
   "DB_Field_Field{2,15}_HMI_Visualization" : USInt = PLC DB_Field.Field[2,15].HMI_Visualization AT %DB1.DBW0, 100 ms
   "DB_Field_Field{2,16}_HMI_Visualization" : USInt = PLC DB_Field.Field[2,16].HMI_Visualization AT %DB1.DBW0, 100 ms
   "DB_Field_Field{2,17}_HMI_Visualization" : USInt = PLC DB_Field.Field[2,17].HMI_Visualization AT %DB1.DBW0, 100 ms
   "DB_Field_Field{2,18}_HMI_Visualization" : USInt = PLC DB_Field.Field[2,18].HMI_Visualization AT %DB1.DBW0, 100 ms
   "DB_Field_Field{2,19}_HMI_Visualization" : USInt = PLC DB_Field.Field[2,19].HMI_Visualization AT %DB1.DBW0, 100 ms
   "DB_Field_Field{2,20}_HMI_Visualization" : USInt = PLC DB_Field.Field[2,20].HMI_Visualization AT %DB1.DBW0, 100 ms
   "DB_Field_Field{3,1}_HMI_Visualization" : USInt = PLC DB_Field.Field[3,1].HMI_Visualization AT %DB1.DBW0, 100 ms
   "DB_Field_Field{3,2}_HMI_Visualization" : USInt = PLC DB_Field.Field[3,2].HMI_Visualization AT %DB1.DBW0, 100 ms
   "DB_Field_Field{3,3}_HMI_Visualization" : USInt = PLC DB_Field.Field[3,3].HMI_Visualization AT %DB1.DBW0, 100 ms
   "DB_Field_Field{3,4}_HMI_Visualization" : USInt = PLC DB_Field.Field[3,4].HMI_Visualization AT %DB1.DBW0, 100 ms
   "DB_Field_Field{3,5}_HMI_Visualization" : USInt = PLC DB_Field.Field[3,5].HMI_Visualization AT %DB1.DBW0, 100 ms
   "DB_Field_Field{3,6}_HMI_Visualization" : USInt = PLC DB_Field.Field[3,6].HMI_Visualization AT %DB1.DBW0, 100 ms
   "DB_Field_Field{3,7}_HMI_Visualization" : USInt = PLC DB_Field.Field[3,7].HMI_Visualization AT %DB1.DBW0, 100 ms
   "DB_Field_Field{3,8}_HMI_Visualization" : USInt = PLC DB_Field.Field[3,8].HMI_Visualization AT %DB1.DBW0, 100 ms
   "DB_Field_Field{3,9}_HMI_Visualization" : USInt = PLC DB_Field.Field[3,9].HMI_Visualization AT %DB1.DBW0, 100 ms
   "DB_Field_Field{3,10}_HMI_Visualization" : USInt = PLC DB_Field.Field[3,10].HMI_Visualization AT %DB1.DBW0, 100 ms
   "DB_Field_Field{3,11}_HMI_Visualization" : USInt = PLC DB_Field.Field[3,11].HMI_Visualization AT %DB1.DBW0, 100 ms
   "DB_Field_Field{3,12}_HMI_Visualization" : USInt = PLC DB_Field.Field[3,12].HMI_Visualization AT %DB1.DBW0, 100 ms
   "DB_Field_Field{3,13}_HMI_Visualization" : USInt = PLC DB_Field.Field[3,13].HMI_Visualization AT %DB1.DBW0, 100 ms
   "DB_Field_Field{3,14}_HMI_Visualization" : USInt = PLC DB_Field.Field[3,14].HMI_Visualization AT %DB1.DBW0, 100 ms
   "DB_Field_Field{3,15}_HMI_Visualization" : USInt = PLC DB_Field.Field[3,15].HMI_Visualization AT %DB1.DBW0, 100 ms
   "DB_Field_Field{3,16}_HMI_Visualization" : USInt = PLC DB_Field.Field[3,16].HMI_Visualization AT %DB1.DBW0, 100 ms
   "DB_Field_Field{3,17}_HMI_Visualization" : USInt = PLC DB_Field.Field[3,17].HMI_Visualization AT %DB1.DBW0, 100 ms
   "DB_Field_Field{3,18}_HMI_Visualization" : USInt = PLC DB_Field.Field[3,18].HMI_Visualization AT %DB1.DBW0, 100 ms
   "DB_Field_Field{3,19}_HMI_Visualization" : USInt = PLC DB_Field.Field[3,19].HMI_Visualization AT %DB1.DBW0, 100 ms
   "DB_Field_Field{3,20}_HMI_Visualization" : USInt = PLC DB_Field.Field[3,20].HMI_Visualization AT %DB1.DBW0, 100 ms
   "DB_Field_Field{4,1}_HMI_Visualization" : USInt = PLC DB_Field.Field[4,1].HMI_Visualization AT %DB1.DBW0, 100 ms
   "DB_Field_Field{4,2}_HMI_Visualization" : USInt = PLC DB_Field.Field[4,2].HMI_Visualization AT %DB1.DBW0, 100 ms
   "DB_Field_Field{4,3}_HMI_Visualization" : USInt = PLC DB_Field.Field[4,3].HMI_Visualization AT %DB1.DBW0, 100 ms
   "DB_Field_Field{4,4}_HMI_Visualization" : USInt = PLC DB_Field.Field[4,4].HMI_Visualization AT %DB1.DBW0, 100 ms
   "DB_Field_Field{4,5}_HMI_Visualization" : USInt = PLC DB_Field.Field[4,5].HMI_Visualization AT %DB1.DBW0, 100 ms
   "DB_Field_Field{4,6}_HMI_Visualization" : USInt = PLC DB_Field.Field[4,6].HMI_Visualization AT %DB1.DBW0, 100 ms
   "DB_Field_Field{4,7}_HMI_Visualization" : USInt = PLC DB_Field.Field[4,7].HMI_Visualization AT %DB1.DBW0, 100 ms
   "DB_Field_Field{4,8}_HMI_Visualization" : USInt = PLC DB_Field.Field[4,8].HMI_Visualization AT %DB1.DBW0, 100 ms
   "DB_Field_Field{4,9}_HMI_Visualization" : USInt = PLC DB_Field.Field[4,9].HMI_Visualization AT %DB1.DBW0, 100 ms
   "DB_Field_Field{4,10}_HMI_Visualization" : USInt = PLC DB_Field.Field[4,10].HMI_Visualization AT %DB1.DBW0, 100 ms
   "DB_Field_Field{4,11}_HMI_Visualization" : USInt = PLC DB_Field.Field[4,11].HMI_Visualization AT %DB1.DBW0, 100 ms
   "DB_Field_Field{4,12}_HMI_Visualization" : USInt = PLC DB_Field.Field[4,12].HMI_Visualization AT %DB1.DBW0, 100 ms
   "DB_Field_Field{4,13}_HMI_Visualization" : USInt = PLC DB_Field.Field[4,13].HMI_Visualization AT %DB1.DBW0, 100 ms
   "DB_Field_Field{4,14}_HMI_Visualization" : USInt = PLC DB_Field.Field[4,14].HMI_Visualization AT %DB1.DBW0, 100 ms
   "DB_Field_Field{4,15}_HMI_Visualization" : USInt = PLC DB_Field.Field[4,15].HMI_Visualization AT %DB1.DBW0, 100 ms
   "DB_Field_Field{4,16}_HMI_Visualization" : USInt = PLC DB_Field.Field[4,16].HMI_Visualization AT %DB1.DBW0, 100 ms
   "DB_Field_Field{4,17}_HMI_Visualization" : USInt = PLC DB_Field.Field[4,17].HMI_Visualization AT %DB1.DBW0, 100 ms
   "DB_Field_Field{4,18}_HMI_Visualization" : USInt = PLC DB_Field.Field[4,18].HMI_Visualization AT %DB1.DBW0, 100 ms
   "DB_Field_Field{4,19}_HMI_Visualization" : USInt = PLC DB_Field.Field[4,19].HMI_Visualization AT %DB1.DBW0, 100 ms
   "DB_Field_Field{4,20}_HMI_Visualization" : USInt = PLC DB_Field.Field[4,20].HMI_Visualization AT %DB1.DBW0, 100 ms
   "DB_Field_Field{5,1}_HMI_Visualization" : USInt = PLC DB_Field.Field[5,1].HMI_Visualization AT %DB1.DBW0, 100 ms
   "DB_Field_Field{5,2}_HMI_Visualization" : USInt = PLC DB_Field.Field[5,2].HMI_Visualization AT %DB1.DBW0, 100 ms
   "DB_Field_Field{5,3}_HMI_Visualization" : USInt = PLC DB_Field.Field[5,3].HMI_Visualization AT %DB1.DBW0, 100 ms
   "DB_Field_Field{5,4}_HMI_Visualization" : USInt = PLC DB_Field.Field[5,4].HMI_Visualization AT %DB1.DBW0, 100 ms
   "DB_Field_Field{5,5}_HMI_Visualization" : USInt = PLC DB_Field.Field[5,5].HMI_Visualization AT %DB1.DBW0, 100 ms
   "DB_Field_Field{5,6}_HMI_Visualization" : USInt = PLC DB_Field.Field[5,6].HMI_Visualization AT %DB1.DBW0, 100 ms
   "DB_Field_Field{5,7}_HMI_Visualization" : USInt = PLC DB_Field.Field[5,7].HMI_Visualization AT %DB1.DBW0, 100 ms
   "DB_Field_Field{5,8}_HMI_Visualization" : USInt = PLC DB_Field.Field[5,8].HMI_Visualization AT %DB1.DBW0, 100 ms
   "DB_Field_Field{5,9}_HMI_Visualization" : USInt = PLC DB_Field.Field[5,9].HMI_Visualization AT %DB1.DBW0, 100 ms
   "DB_Field_Field{5,10}_HMI_Visualization" : USInt = PLC DB_Field.Field[5,10].HMI_Visualization AT %DB1.DBW0, 100 ms
   "DB_Field_Field{5,11}_HMI_Visualization" : USInt = PLC DB_Field.Field[5,11].HMI_Visualization AT %DB1.DBW0, 100 ms
   "DB_Field_Field{5,12}_HMI_Visualization" : USInt = PLC DB_Field.Field[5,12].HMI_Visualization AT %DB1.DBW0, 100 ms
   "DB_Field_Field{5,13}_HMI_Visualization" : USInt = PLC DB_Field.Field[5,13].HMI_Visualization AT %DB1.DBW0, 100 ms
   "DB_Field_Field{5,14}_HMI_Visualization" : USInt = PLC DB_Field.Field[5,14].HMI_Visualization AT %DB1.DBW0, 100 ms
   "DB_Field_Field{5,15}_HMI_Visualization" : USInt = PLC DB_Field.Field[5,15].HMI_Visualization AT %DB1.DBW0, 100 ms
   "DB_Field_Field{5,16}_HMI_Visualization" : USInt = PLC DB_Field.Field[5,16].HMI_Visualization AT %DB1.DBW0, 100 ms
   "DB_Field_Field{5,17}_HMI_Visualization" : USInt = PLC DB_Field.Field[5,17].HMI_Visualization AT %DB1.DBW0, 100 ms
   "DB_Field_Field{5,18}_HMI_Visualization" : USInt = PLC DB_Field.Field[5,18].HMI_Visualization AT %DB1.DBW0, 100 ms
   "DB_Field_Field{5,19}_HMI_Visualization" : USInt = PLC DB_Field.Field[5,19].HMI_Visualization AT %DB1.DBW0, 100 ms
   "DB_Field_Field{5,20}_HMI_Visualization" : USInt = PLC DB_Field.Field[5,20].HMI_Visualization AT %DB1.DBW0, 100 ms
   "DB_Field_Field{6,1}_HMI_Visualization" : USInt = PLC DB_Field.Field[6,1].HMI_Visualization AT %DB1.DBW0, 100 ms
   "DB_Field_Field{6,2}_HMI_Visualization" : USInt = PLC DB_Field.Field[6,2].HMI_Visualization AT %DB1.DBW0, 100 ms
   "DB_Field_Field{6,3}_HMI_Visualization" : USInt = PLC DB_Field.Field[6,3].HMI_Visualization AT %DB1.DBW0, 100 ms
   "DB_Field_Field{6,4}_HMI_Visualization" : USInt = PLC DB_Field.Field[6,4].HMI_Visualization AT %DB1.DBW0, 100 ms
   "DB_Field_Field{6,5}_HMI_Visualization" : USInt = PLC DB_Field.Field[6,5].HMI_Visualization AT %DB1.DBW0, 100 ms
   "DB_Field_Field{6,6}_HMI_Visualization" : USInt = PLC DB_Field.Field[6,6].HMI_Visualization AT %DB1.DBW0, 100 ms
   "DB_Field_Field{6,7}_HMI_Visualization" : USInt = PLC DB_Field.Field[6,7].HMI_Visualization AT %DB1.DBW0, 100 ms
   "DB_Field_Field{6,8}_HMI_Visualization" : USInt = PLC DB_Field.Field[6,8].HMI_Visualization AT %DB1.DBW0, 100 ms
   "DB_Field_Field{6,9}_HMI_Visualization" : USInt = PLC DB_Field.Field[6,9].HMI_Visualization AT %DB1.DBW0, 100 ms
   "DB_Field_Field{6,10}_HMI_Visualization" : USInt = PLC DB_Field.Field[6,10].HMI_Visualization AT %DB1.DBW0, 100 ms
   "DB_Field_Field{6,11}_HMI_Visualization" : USInt = PLC DB_Field.Field[6,11].HMI_Visualization AT %DB1.DBW0, 100 ms
   "DB_Field_Field{6,12}_HMI_Visualization" : USInt = PLC DB_Field.Field[6,12].HMI_Visualization AT %DB1.DBW0, 100 ms
   "DB_Field_Field{6,13}_HMI_Visualization" : USInt = PLC DB_Field.Field[6,13].HMI_Visualization AT %DB1.DBW0, 100 ms
   "DB_Field_Field{6,14}_HMI_Visualization" : USInt = PLC DB_Field.Field[6,14].HMI_Visualization AT %DB1.DBW0, 100 ms
   "DB_Field_Field{6,15}_HMI_Visualization" : USInt = PLC DB_Field.Field[6,15].HMI_Visualization AT %DB1.DBW0, 100 ms
   "DB_Field_Field{6,16}_HMI_Visualization" : USInt = PLC DB_Field.Field[6,16].HMI_Visualization AT %DB1.DBW0, 100 ms
   "DB_Field_Field{6,17}_HMI_Visualization" : USInt = PLC DB_Field.Field[6,17].HMI_Visualization AT %DB1.DBW0, 100 ms
   "DB_Field_Field{6,18}_HMI_Visualization" : USInt = PLC DB_Field.Field[6,18].HMI_Visualization AT %DB1.DBW0, 100 ms
   "DB_Field_Field{6,19}_HMI_Visualization" : USInt = PLC DB_Field.Field[6,19].HMI_Visualization AT %DB1.DBW0, 100 ms
   "DB_Field_Field{6,20}_HMI_Visualization" : USInt = PLC DB_Field.Field[6,20].HMI_Visualization AT %DB1.DBW0, 100 ms
   "DB_Field_Field{7,1}_HMI_Visualization" : USInt = PLC DB_Field.Field[7,1].HMI_Visualization AT %DB1.DBW0, 100 ms
   "DB_Field_Field{7,2}_HMI_Visualization" : USInt = PLC DB_Field.Field[7,2].HMI_Visualization AT %DB1.DBW0, 100 ms
   "DB_Field_Field{7,3}_HMI_Visualization" : USInt = PLC DB_Field.Field[7,3].HMI_Visualization AT %DB1.DBW0, 100 ms
   "DB_Field_Field{7,4}_HMI_Visualization" : USInt = PLC DB_Field.Field[7,4].HMI_Visualization AT %DB1.DBW0, 100 ms
   "DB_Field_Field{7,5}_HMI_Visualization" : USInt = PLC DB_Field.Field[7,5].HMI_Visualization AT %DB1.DBW0, 100 ms
   "DB_Field_Field{7,6}_HMI_Visualization" : USInt = PLC DB_Field.Field[7,6].HMI_Visualization AT %DB1.DBW0, 100 ms
   "DB_Field_Field{7,7}_HMI_Visualization" : USInt = PLC DB_Field.Field[7,7].HMI_Visualization AT %DB1.DBW0, 100 ms
   "DB_Field_Field{7,8}_HMI_Visualization" : USInt = PLC DB_Field.Field[7,8].HMI_Visualization AT %DB1.DBW0, 100 ms
   "DB_Field_Field{7,9}_HMI_Visualization" : USInt = PLC DB_Field.Field[7,9].HMI_Visualization AT %DB1.DBW0, 100 ms
   "DB_Field_Field{7,10}_HMI_Visualization" : USInt = PLC DB_Field.Field[7,10].HMI_Visualization AT %DB1.DBW0, 100 ms
   "DB_Field_Field{7,11}_HMI_Visualization" : USInt = PLC DB_Field.Field[7,11].HMI_Visualization AT %DB1.DBW0, 100 ms
   "DB_Field_Field{7,12}_HMI_Visualization" : USInt = PLC DB_Field.Field[7,12].HMI_Visualization AT %DB1.DBW0, 100 ms
   "DB_Field_Field{7,13}_HMI_Visualization" : USInt = PLC DB_Field.Field[7,13].HMI_Visualization AT %DB1.DBW0, 100 ms
   "DB_Field_Field{7,14}_HMI_Visualization" : USInt = PLC DB_Field.Field[7,14].HMI_Visualization AT %DB1.DBW0, 100 ms
   "DB_Field_Field{7,15}_HMI_Visualization" : USInt = PLC DB_Field.Field[7,15].HMI_Visualization AT %DB1.DBW0, 100 ms
   "DB_Field_Field{7,16}_HMI_Visualization" : USInt = PLC DB_Field.Field[7,16].HMI_Visualization AT %DB1.DBW0, 100 ms
   "DB_Field_Field{7,17}_HMI_Visualization" : USInt = PLC DB_Field.Field[7,17].HMI_Visualization AT %DB1.DBW0, 100 ms
   "DB_Field_Field{7,18}_HMI_Visualization" : USInt = PLC DB_Field.Field[7,18].HMI_Visualization AT %DB1.DBW0, 100 ms
   "DB_Field_Field{7,19}_HMI_Visualization" : USInt = PLC DB_Field.Field[7,19].HMI_Visualization AT %DB1.DBW0, 100 ms
   "DB_Field_Field{7,20}_HMI_Visualization" : USInt = PLC DB_Field.Field[7,20].HMI_Visualization AT %DB1.DBW0, 100 ms
   "DB_Field_Field{8,1}_HMI_Visualization" : USInt = PLC DB_Field.Field[8,1].HMI_Visualization AT %DB1.DBW0, 100 ms
   "DB_Field_Field{8,2}_HMI_Visualization" : USInt = PLC DB_Field.Field[8,2].HMI_Visualization AT %DB1.DBW0, 100 ms
   "DB_Field_Field{8,3}_HMI_Visualization" : USInt = PLC DB_Field.Field[8,3].HMI_Visualization AT %DB1.DBW0, 100 ms
   "DB_Field_Field{8,4}_HMI_Visualization" : USInt = PLC DB_Field.Field[8,4].HMI_Visualization AT %DB1.DBW0, 100 ms
   "DB_Field_Field{8,5}_HMI_Visualization" : USInt = PLC DB_Field.Field[8,5].HMI_Visualization AT %DB1.DBW0, 100 ms
   "DB_Field_Field{8,6}_HMI_Visualization" : USInt = PLC DB_Field.Field[8,6].HMI_Visualization AT %DB1.DBW0, 100 ms
   "DB_Field_Field{8,7}_HMI_Visualization" : USInt = PLC DB_Field.Field[8,7].HMI_Visualization AT %DB1.DBW0, 100 ms
   "DB_Field_Field{8,8}_HMI_Visualization" : USInt = PLC DB_Field.Field[8,8].HMI_Visualization AT %DB1.DBW0, 100 ms
   "DB_Field_Field{8,9}_HMI_Visualization" : USInt = PLC DB_Field.Field[8,9].HMI_Visualization AT %DB1.DBW0, 100 ms
   "DB_Field_Field{8,10}_HMI_Visualization" : USInt = PLC DB_Field.Field[8,10].HMI_Visualization AT %DB1.DBW0, 100 ms
   "DB_Field_Field{8,11}_HMI_Visualization" : USInt = PLC DB_Field.Field[8,11].HMI_Visualization AT %DB1.DBW0, 100 ms
   "DB_Field_Field{8,12}_HMI_Visualization" : USInt = PLC DB_Field.Field[8,12].HMI_Visualization AT %DB1.DBW0, 100 ms
   "DB_Field_Field{8,13}_HMI_Visualization" : USInt = PLC DB_Field.Field[8,13].HMI_Visualization AT %DB1.DBW0, 100 ms
   "DB_Field_Field{8,14}_HMI_Visualization" : USInt = PLC DB_Field.Field[8,14].HMI_Visualization AT %DB1.DBW0, 100 ms
   "DB_Field_Field{8,15}_HMI_Visualization" : USInt = PLC DB_Field.Field[8,15].HMI_Visualization AT %DB1.DBW0, 100 ms
   "DB_Field_Field{8,16}_HMI_Visualization" : USInt = PLC DB_Field.Field[8,16].HMI_Visualization AT %DB1.DBW0, 100 ms
   "DB_Field_Field{8,17}_HMI_Visualization" : USInt = PLC DB_Field.Field[8,17].HMI_Visualization AT %DB1.DBW0, 100 ms
   "DB_Field_Field{8,18}_HMI_Visualization" : USInt = PLC DB_Field.Field[8,18].HMI_Visualization AT %DB1.DBW0, 100 ms
   "DB_Field_Field{8,19}_HMI_Visualization" : USInt = PLC DB_Field.Field[8,19].HMI_Visualization AT %DB1.DBW0, 100 ms
   "DB_Field_Field{8,20}_HMI_Visualization" : USInt = PLC DB_Field.Field[8,20].HMI_Visualization AT %DB1.DBW0, 100 ms
   "DB_Field_Field{9,1}_HMI_Visualization" : USInt = PLC DB_Field.Field[9,1].HMI_Visualization AT %DB1.DBW0, 100 ms
   "DB_Field_Field{9,2}_HMI_Visualization" : USInt = PLC DB_Field.Field[9,2].HMI_Visualization AT %DB1.DBW0, 100 ms
   "DB_Field_Field{9,3}_HMI_Visualization" : USInt = PLC DB_Field.Field[9,3].HMI_Visualization AT %DB1.DBW0, 100 ms
   "DB_Field_Field{9,4}_HMI_Visualization" : USInt = PLC DB_Field.Field[9,4].HMI_Visualization AT %DB1.DBW0, 100 ms
   "DB_Field_Field{9,5}_HMI_Visualization" : USInt = PLC DB_Field.Field[9,5].HMI_Visualization AT %DB1.DBW0, 100 ms
   "DB_Field_Field{9,6}_HMI_Visualization" : USInt = PLC DB_Field.Field[9,6].HMI_Visualization AT %DB1.DBW0, 100 ms
   "DB_Field_Field{9,7}_HMI_Visualization" : USInt = PLC DB_Field.Field[9,7].HMI_Visualization AT %DB1.DBW0, 100 ms
   "DB_Field_Field{9,8}_HMI_Visualization" : USInt = PLC DB_Field.Field[9,8].HMI_Visualization AT %DB1.DBW0, 100 ms
   "DB_Field_Field{9,9}_HMI_Visualization" : USInt = PLC DB_Field.Field[9,9].HMI_Visualization AT %DB1.DBW0, 100 ms
   "DB_Field_Field{9,10}_HMI_Visualization" : USInt = PLC DB_Field.Field[9,10].HMI_Visualization AT %DB1.DBW0, 100 ms
   "DB_Field_Field{9,11}_HMI_Visualization" : USInt = PLC DB_Field.Field[9,11].HMI_Visualization AT %DB1.DBW0, 100 ms
   "DB_Field_Field{9,12}_HMI_Visualization" : USInt = PLC DB_Field.Field[9,12].HMI_Visualization AT %DB1.DBW0, 100 ms
   "DB_Field_Field{9,13}_HMI_Visualization" : USInt = PLC DB_Field.Field[9,13].HMI_Visualization AT %DB1.DBW0, 100 ms
   "DB_Field_Field{9,14}_HMI_Visualization" : USInt = PLC DB_Field.Field[9,14].HMI_Visualization AT %DB1.DBW0, 100 ms
   "DB_Field_Field{9,15}_HMI_Visualization" : USInt = PLC DB_Field.Field[9,15].HMI_Visualization AT %DB1.DBW0, 100 ms
   "DB_Field_Field{9,16}_HMI_Visualization" : USInt = PLC DB_Field.Field[9,16].HMI_Visualization AT %DB1.DBW0, 100 ms
   "DB_Field_Field{9,17}_HMI_Visualization" : USInt = PLC DB_Field.Field[9,17].HMI_Visualization AT %DB1.DBW0, 100 ms
   "DB_Field_Field{9,18}_HMI_Visualization" : USInt = PLC DB_Field.Field[9,18].HMI_Visualization AT %DB1.DBW0, 100 ms
   "DB_Field_Field{9,19}_HMI_Visualization" : USInt = PLC DB_Field.Field[9,19].HMI_Visualization AT %DB1.DBW0, 100 ms
   "DB_Field_Field{9,20}_HMI_Visualization" : USInt = PLC DB_Field.Field[9,20].HMI_Visualization AT %DB1.DBW0, 100 ms
   "DB_Field_Field{10,1}_HMI_Visualization" : USInt = PLC DB_Field.Field[10,1].HMI_Visualization AT %DB1.DBW0, 100 ms
   "DB_Field_Field{10,2}_HMI_Visualization" : USInt = PLC DB_Field.Field[10,2].HMI_Visualization AT %DB1.DBW0, 100 ms
   "DB_Field_Field{10,3}_HMI_Visualization" : USInt = PLC DB_Field.Field[10,3].HMI_Visualization AT %DB1.DBW0, 100 ms
   "DB_Field_Field{10,4}_HMI_Visualization" : USInt = PLC DB_Field.Field[10,4].HMI_Visualization AT %DB1.DBW0, 100 ms
   "DB_Field_Field{10,5}_HMI_Visualization" : USInt = PLC DB_Field.Field[10,5].HMI_Visualization AT %DB1.DBW0, 100 ms
   "DB_Field_Field{10,6}_HMI_Visualization" : USInt = PLC DB_Field.Field[10,6].HMI_Visualization AT %DB1.DBW0, 100 ms
   "DB_Field_Field{10,7}_HMI_Visualization" : USInt = PLC DB_Field.Field[10,7].HMI_Visualization AT %DB1.DBW0, 100 ms
   "DB_Field_Field{10,8}_HMI_Visualization" : USInt = PLC DB_Field.Field[10,8].HMI_Visualization AT %DB1.DBW0, 100 ms
   "DB_Field_Field{10,9}_HMI_Visualization" : USInt = PLC DB_Field.Field[10,9].HMI_Visualization AT %DB1.DBW0, 100 ms
   "DB_Field_Field{10,10}_HMI_Visualization" : USInt = PLC DB_Field.Field[10,10].HMI_Visualization AT %DB1.DBW0, 100 ms
   "DB_Field_Field{10,11}_HMI_Visualization" : USInt = PLC DB_Field.Field[10,11].HMI_Visualization AT %DB1.DBW0, 100 ms
   "DB_Field_Field{10,12}_HMI_Visualization" : USInt = PLC DB_Field.Field[10,12].HMI_Visualization AT %DB1.DBW0, 100 ms
   "DB_Field_Field{10,13}_HMI_Visualization" : USInt = PLC DB_Field.Field[10,13].HMI_Visualization AT %DB1.DBW0, 100 ms
   "DB_Field_Field{10,14}_HMI_Visualization" : USInt = PLC DB_Field.Field[10,14].HMI_Visualization AT %DB1.DBW0, 100 ms
   "DB_Field_Field{10,15}_HMI_Visualization" : USInt = PLC DB_Field.Field[10,15].HMI_Visualization AT %DB1.DBW0, 100 ms
   "DB_Field_Field{10,16}_HMI_Visualization" : USInt = PLC DB_Field.Field[10,16].HMI_Visualization AT %DB1.DBW0, 100 ms
   "DB_Field_Field{10,17}_HMI_Visualization" : USInt = PLC DB_Field.Field[10,17].HMI_Visualization AT %DB1.DBW0, 100 ms
   "DB_Field_Field{10,18}_HMI_Visualization" : USInt = PLC DB_Field.Field[10,18].HMI_Visualization AT %DB1.DBW0, 100 ms
   "DB_Field_Field{10,19}_HMI_Visualization" : USInt = PLC DB_Field.Field[10,19].HMI_Visualization AT %DB1.DBW0, 100 ms
   "DB_Field_Field{10,20}_HMI_Visualization" : USInt = PLC DB_Field.Field[10,20].HMI_Visualization AT %DB1.DBW0, 100 ms
   "DB_Commands_Cmd_SnakeLeft" : Bool = PLC DB_Commands.Cmd.SnakeLeft, 1 s
   "DB_Commands_Cmd_SnakeRight" : Bool = PLC DB_Commands.Cmd.SnakeRight, 1 s
   "DB_Commands_Cmd_SnakeUp" : Bool = PLC DB_Commands.Cmd.SnakeUp, 1 s
   "DB_Commands_Cmd_SnakeDown" : Bool = PLC DB_Commands.Cmd.SnakeDown, 1 s
   "DB_Commands_Sts_GameActive" : Bool = PLC DB_Commands.Sts.GameActive, 1 s
   "DB_Commands_Points_Actual" : UDInt = PLC DB_Commands.Points.Actual, 1 s
   "DB_Commands_Points_BestGame" : UDInt = PLC DB_Commands.Points.BestGame, 1 s
   "DB_Commands_Cmd_Stop" : Bool = PLC DB_Commands.Cmd.Stop, 1 s
   "DB_Commands_Sts_PauseActive" : Bool = PLC DB_Commands.Sts.PauseActive, 1 s
   "DB_Commands_Cmd_Pause" : Bool = PLC DB_Commands.Cmd.Pause, 1 s
   "DB_Commands_Cmd_Start" : Bool = PLC DB_Commands.Cmd.Start, 1 s
   "DB_Commands_Cmd_Speed" : Real = PLC DB_Commands.Cmd.Speed, 1 s
   "DB_Commands_Sts_SnakeLength" : UDInt = PLC DB_Commands.Sts.SnakeLength, 1 s

text list "Elenco testi_Nome della pagina": 1 'Pagina base'

screen "Pagina base" 1920x1020, template "Modello_1"
   on GenerateScreen: SetTag("Variabile_Numero di pagina", 1)
   Rectangle "Rettangolo_1" at 25,665 size 72x72
      Appearance <- "DB_Field_Field{1,1}_HMI_Visualization"
   Rectangle "Rettangolo_2" at 97,665 size 72x72
      Appearance <- "DB_Field_Field{1,2}_HMI_Visualization"
   Rectangle "Rettangolo_3" at 168,665 size 72x72
      Appearance <- "DB_Field_Field{1,3}_HMI_Visualization"
   Rectangle "Rettangolo_4" at 240,665 size 72x72
      Appearance <- "DB_Field_Field{1,4}_HMI_Visualization"
   Rectangle "Rettangolo_5" at 311,665 size 72x72
      Appearance <- "DB_Field_Field{1,5}_HMI_Visualization"
   Rectangle "Rettangolo_6" at 383,665 size 72x72
      Appearance <- "DB_Field_Field{1,6}_HMI_Visualization"
   Rectangle "Rettangolo_7" at 454,665 size 72x72
      Appearance <- "DB_Field_Field{1,7}_HMI_Visualization"
   Rectangle "Rettangolo_8" at 526,665 size 72x72
      Appearance <- "DB_Field_Field{1,8}_HMI_Visualization"
   Rectangle "Rettangolo_9" at 598,665 size 72x72
      Appearance <- "DB_Field_Field{1,9}_HMI_Visualization"
   Rectangle "Rettangolo_10" at 670,665 size 72x72
      Appearance <- "DB_Field_Field{1,10}_HMI_Visualization"
   Rectangle "Rettangolo_11" at 741,665 size 72x72
      Appearance <- "DB_Field_Field{1,11}_HMI_Visualization"
   Rectangle "Rettangolo_12" at 813,665 size 72x72
      Appearance <- "DB_Field_Field{1,12}_HMI_Visualization"
   Rectangle "Rettangolo_13" at 884,665 size 72x72
      Appearance <- "DB_Field_Field{1,13}_HMI_Visualization"
   Rectangle "Rettangolo_14" at 956,665 size 72x72
      Appearance <- "DB_Field_Field{1,14}_HMI_Visualization"
   Rectangle "Rettangolo_15" at 1027,665 size 72x72
      Appearance <- "DB_Field_Field{1,15}_HMI_Visualization"
   Rectangle "Rettangolo_16" at 1099,665 size 72x72
      Appearance <- "DB_Field_Field{1,16}_HMI_Visualization"
   Rectangle "Rettangolo_17" at 1170,665 size 72x72
      Appearance <- "DB_Field_Field{1,17}_HMI_Visualization"
   Rectangle "Rettangolo_18" at 1242,665 size 72x72
      Appearance <- "DB_Field_Field{1,18}_HMI_Visualization"
   Rectangle "Rettangolo_19" at 1314,665 size 72x72
      Appearance <- "DB_Field_Field{1,19}_HMI_Visualization"
   Rectangle "Rettangolo_20" at 1386,665 size 72x72
      Appearance <- "DB_Field_Field{1,20}_HMI_Visualization"
   Rectangle "Rettangolo_21" at 25,593 size 72x72
      Appearance <- "DB_Field_Field{2,1}_HMI_Visualization"
   Rectangle "Rettangolo_22" at 97,593 size 72x72
      Appearance <- "DB_Field_Field{2,2}_HMI_Visualization"
   Rectangle "Rettangolo_23" at 168,593 size 72x72
      Appearance <- "DB_Field_Field{2,3}_HMI_Visualization"
   Rectangle "Rettangolo_24" at 240,593 size 72x72
      Appearance <- "DB_Field_Field{2,4}_HMI_Visualization"
   Rectangle "Rettangolo_25" at 311,593 size 72x72
      Appearance <- "DB_Field_Field{2,5}_HMI_Visualization"
   Rectangle "Rettangolo_26" at 383,593 size 72x72
      Appearance <- "DB_Field_Field{2,6}_HMI_Visualization"
   Rectangle "Rettangolo_27" at 454,593 size 72x72
      Appearance <- "DB_Field_Field{2,7}_HMI_Visualization"
   Rectangle "Rettangolo_28" at 526,593 size 72x72
      Appearance <- "DB_Field_Field{2,8}_HMI_Visualization"
   Rectangle "Rettangolo_29" at 598,593 size 72x72
      Appearance <- "DB_Field_Field{2,9}_HMI_Visualization"
   Rectangle "Rettangolo_30" at 670,593 size 72x72
      Appearance <- "DB_Field_Field{2,10}_HMI_Visualization"
   Rectangle "Rettangolo_31" at 741,593 size 72x72
      Appearance <- "DB_Field_Field{2,11}_HMI_Visualization"
   Rectangle "Rettangolo_32" at 813,593 size 72x72
      Appearance <- "DB_Field_Field{2,12}_HMI_Visualization"
   Rectangle "Rettangolo_33" at 884,593 size 72x72
      Appearance <- "DB_Field_Field{2,13}_HMI_Visualization"
   Rectangle "Rettangolo_34" at 956,593 size 72x72
      Appearance <- "DB_Field_Field{2,14}_HMI_Visualization"
   Rectangle "Rettangolo_35" at 1027,593 size 72x72
      Appearance <- "DB_Field_Field{2,15}_HMI_Visualization"
   Rectangle "Rettangolo_36" at 1099,593 size 72x72
      Appearance <- "DB_Field_Field{2,16}_HMI_Visualization"
   Rectangle "Rettangolo_37" at 1170,593 size 72x72
      Appearance <- "DB_Field_Field{2,17}_HMI_Visualization"
   Rectangle "Rettangolo_38" at 1242,593 size 72x72
      Appearance <- "DB_Field_Field{2,18}_HMI_Visualization"
   Rectangle "Rettangolo_39" at 1314,593 size 72x72
      Appearance <- "DB_Field_Field{2,19}_HMI_Visualization"
   Rectangle "Rettangolo_40" at 1386,593 size 72x72
      Appearance <- "DB_Field_Field{2,20}_HMI_Visualization"
   Rectangle "Rettangolo_41" at 25,520 size 72x72
      Appearance <- "DB_Field_Field{3,1}_HMI_Visualization"
   Rectangle "Rettangolo_42" at 97,520 size 72x72
      Appearance <- "DB_Field_Field{3,2}_HMI_Visualization"
   Rectangle "Rettangolo_43" at 168,520 size 72x72
      Appearance <- "DB_Field_Field{3,3}_HMI_Visualization"
   Rectangle "Rettangolo_44" at 240,520 size 72x72
      Appearance <- "DB_Field_Field{3,4}_HMI_Visualization"
   Rectangle "Rettangolo_45" at 311,520 size 72x72
      Appearance <- "DB_Field_Field{3,5}_HMI_Visualization"
   Rectangle "Rettangolo_46" at 383,520 size 72x72
      Appearance <- "DB_Field_Field{3,6}_HMI_Visualization"
   Rectangle "Rettangolo_47" at 454,520 size 72x72
      Appearance <- "DB_Field_Field{3,7}_HMI_Visualization"
   Rectangle "Rettangolo_48" at 526,520 size 72x72
      Appearance <- "DB_Field_Field{3,8}_HMI_Visualization"
   Rectangle "Rettangolo_49" at 598,520 size 72x72
      Appearance <- "DB_Field_Field{3,9}_HMI_Visualization"
   Rectangle "Rettangolo_50" at 670,520 size 72x72
      Appearance <- "DB_Field_Field{3,10}_HMI_Visualization"
   Rectangle "Rettangolo_51" at 741,520 size 72x72
      Appearance <- "DB_Field_Field{3,11}_HMI_Visualization"
   Rectangle "Rettangolo_52" at 813,520 size 72x72
      Appearance <- "DB_Field_Field{3,12}_HMI_Visualization"
   Rectangle "Rettangolo_53" at 884,520 size 72x72
      Appearance <- "DB_Field_Field{3,13}_HMI_Visualization"
   Rectangle "Rettangolo_54" at 956,520 size 72x72
      Appearance <- "DB_Field_Field{3,14}_HMI_Visualization"
   Rectangle "Rettangolo_55" at 1027,520 size 72x72
      Appearance <- "DB_Field_Field{3,15}_HMI_Visualization"
   Rectangle "Rettangolo_56" at 1099,520 size 72x72
      Appearance <- "DB_Field_Field{3,16}_HMI_Visualization"
   Rectangle "Rettangolo_57" at 1170,520 size 72x72
      Appearance <- "DB_Field_Field{3,17}_HMI_Visualization"
   Rectangle "Rettangolo_58" at 1242,520 size 72x72
      Appearance <- "DB_Field_Field{3,18}_HMI_Visualization"
   Rectangle "Rettangolo_59" at 1314,520 size 72x72
      Appearance <- "DB_Field_Field{3,19}_HMI_Visualization"
   Rectangle "Rettangolo_60" at 1386,520 size 72x72
      Appearance <- "DB_Field_Field{3,20}_HMI_Visualization"
   Rectangle "Rettangolo_61" at 25,448 size 72x72
      Appearance <- "DB_Field_Field{4,1}_HMI_Visualization"
   Rectangle "Rettangolo_62" at 97,448 size 72x72
      Appearance <- "DB_Field_Field{4,2}_HMI_Visualization"
   Rectangle "Rettangolo_63" at 168,448 size 72x72
      Appearance <- "DB_Field_Field{4,3}_HMI_Visualization"
   Rectangle "Rettangolo_64" at 240,448 size 72x72
      Appearance <- "DB_Field_Field{4,4}_HMI_Visualization"
   Rectangle "Rettangolo_65" at 311,448 size 72x72
      Appearance <- "DB_Field_Field{4,5}_HMI_Visualization"
   Rectangle "Rettangolo_66" at 383,448 size 72x72
      Appearance <- "DB_Field_Field{4,6}_HMI_Visualization"
   Rectangle "Rettangolo_67" at 454,448 size 72x72
      Appearance <- "DB_Field_Field{4,7}_HMI_Visualization"
   Rectangle "Rettangolo_68" at 526,448 size 72x72
      Appearance <- "DB_Field_Field{4,8}_HMI_Visualization"
   Rectangle "Rettangolo_69" at 598,448 size 72x72
      Appearance <- "DB_Field_Field{4,9}_HMI_Visualization"
   Rectangle "Rettangolo_70" at 670,448 size 72x72
      Appearance <- "DB_Field_Field{4,10}_HMI_Visualization"
   Rectangle "Rettangolo_71" at 741,448 size 72x72
      Appearance <- "DB_Field_Field{4,11}_HMI_Visualization"
   Rectangle "Rettangolo_72" at 813,448 size 72x72
      Appearance <- "DB_Field_Field{4,12}_HMI_Visualization"
   Rectangle "Rettangolo_73" at 884,448 size 72x72
      Appearance <- "DB_Field_Field{4,13}_HMI_Visualization"
   Rectangle "Rettangolo_74" at 956,448 size 72x72
      Appearance <- "DB_Field_Field{4,14}_HMI_Visualization"
   Rectangle "Rettangolo_75" at 1027,448 size 72x72
      Appearance <- "DB_Field_Field{4,15}_HMI_Visualization"
   Rectangle "Rettangolo_76" at 1099,448 size 72x72
      Appearance <- "DB_Field_Field{4,16}_HMI_Visualization"
   Rectangle "Rettangolo_77" at 1170,448 size 72x72
      Appearance <- "DB_Field_Field{4,17}_HMI_Visualization"
   Rectangle "Rettangolo_78" at 1242,448 size 72x72
      Appearance <- "DB_Field_Field{4,18}_HMI_Visualization"
   Rectangle "Rettangolo_79" at 1314,448 size 72x72
      Appearance <- "DB_Field_Field{4,19}_HMI_Visualization"
   Rectangle "Rettangolo_80" at 1386,448 size 72x72
      Appearance <- "DB_Field_Field{4,20}_HMI_Visualization"
   Rectangle "Rettangolo_81" at 25,375 size 72x72
      Appearance <- "DB_Field_Field{5,1}_HMI_Visualization"
   Rectangle "Rettangolo_82" at 97,375 size 72x72
      Appearance <- "DB_Field_Field{5,2}_HMI_Visualization"
   Rectangle "Rettangolo_83" at 168,375 size 72x72
      Appearance <- "DB_Field_Field{5,3}_HMI_Visualization"
   Rectangle "Rettangolo_84" at 240,375 size 72x72
      Appearance <- "DB_Field_Field{5,4}_HMI_Visualization"
   Rectangle "Rettangolo_85" at 311,375 size 72x72
      Appearance <- "DB_Field_Field{5,5}_HMI_Visualization"
   Rectangle "Rettangolo_86" at 383,375 size 72x72
      Appearance <- "DB_Field_Field{5,6}_HMI_Visualization"
   Rectangle "Rettangolo_87" at 454,375 size 72x72
      Appearance <- "DB_Field_Field{5,7}_HMI_Visualization"
   Rectangle "Rettangolo_88" at 526,375 size 72x72
      Appearance <- "DB_Field_Field{5,8}_HMI_Visualization"
   Rectangle "Rettangolo_89" at 598,375 size 72x72
      Appearance <- "DB_Field_Field{5,9}_HMI_Visualization"
   Rectangle "Rettangolo_90" at 670,375 size 72x72
      Appearance <- "DB_Field_Field{5,10}_HMI_Visualization"
   Rectangle "Rettangolo_91" at 741,375 size 72x72
      Appearance <- "DB_Field_Field{5,11}_HMI_Visualization"
   Rectangle "Rettangolo_92" at 813,375 size 72x72
      Appearance <- "DB_Field_Field{5,12}_HMI_Visualization"
   Rectangle "Rettangolo_93" at 884,375 size 72x72
      Appearance <- "DB_Field_Field{5,13}_HMI_Visualization"
   Rectangle "Rettangolo_94" at 956,375 size 72x72
      Appearance <- "DB_Field_Field{5,14}_HMI_Visualization"
   Rectangle "Rettangolo_95" at 1027,375 size 72x72
      Appearance <- "DB_Field_Field{5,15}_HMI_Visualization"
   Rectangle "Rettangolo_96" at 1099,375 size 72x72
      Appearance <- "DB_Field_Field{5,16}_HMI_Visualization"
   Rectangle "Rettangolo_97" at 1170,375 size 72x72
      Appearance <- "DB_Field_Field{5,17}_HMI_Visualization"
   Rectangle "Rettangolo_98" at 1242,375 size 72x72
      Appearance <- "DB_Field_Field{5,18}_HMI_Visualization"
   Rectangle "Rettangolo_99" at 1314,375 size 72x72
      Appearance <- "DB_Field_Field{5,19}_HMI_Visualization"
   Rectangle "Rettangolo_100" at 1386,375 size 72x72
      Appearance <- "DB_Field_Field{5,20}_HMI_Visualization"
   Rectangle "Rettangolo_101" at 25,303 size 72x72
      Appearance <- "DB_Field_Field{6,1}_HMI_Visualization"
   Rectangle "Rettangolo_102" at 97,303 size 72x72
      Appearance <- "DB_Field_Field{6,2}_HMI_Visualization"
   Rectangle "Rettangolo_103" at 168,303 size 72x72
      Appearance <- "DB_Field_Field{6,3}_HMI_Visualization"
   Rectangle "Rettangolo_104" at 240,303 size 72x72
      Appearance <- "DB_Field_Field{6,4}_HMI_Visualization"
   Rectangle "Rettangolo_105" at 311,303 size 72x72
      Appearance <- "DB_Field_Field{6,5}_HMI_Visualization"
   Rectangle "Rettangolo_106" at 383,303 size 72x72
      Appearance <- "DB_Field_Field{6,6}_HMI_Visualization"
   Rectangle "Rettangolo_107" at 454,303 size 72x72
      Appearance <- "DB_Field_Field{6,7}_HMI_Visualization"
   Rectangle "Rettangolo_108" at 526,303 size 72x72
      Appearance <- "DB_Field_Field{6,8}_HMI_Visualization"
   Rectangle "Rettangolo_109" at 598,303 size 72x72
      Appearance <- "DB_Field_Field{6,9}_HMI_Visualization"
   Rectangle "Rettangolo_110" at 670,303 size 72x72
      Appearance <- "DB_Field_Field{6,10}_HMI_Visualization"
   Rectangle "Rettangolo_111" at 741,303 size 72x72
      Appearance <- "DB_Field_Field{6,11}_HMI_Visualization"
   Rectangle "Rettangolo_112" at 813,303 size 72x72
      Appearance <- "DB_Field_Field{6,12}_HMI_Visualization"
   Rectangle "Rettangolo_113" at 884,303 size 72x72
      Appearance <- "DB_Field_Field{6,13}_HMI_Visualization"
   Rectangle "Rettangolo_114" at 956,303 size 72x72
      Appearance <- "DB_Field_Field{6,14}_HMI_Visualization"
   Rectangle "Rettangolo_115" at 1027,303 size 72x72
      Appearance <- "DB_Field_Field{6,15}_HMI_Visualization"
   Rectangle "Rettangolo_116" at 1099,303 size 72x72
      Appearance <- "DB_Field_Field{6,16}_HMI_Visualization"
   Rectangle "Rettangolo_117" at 1170,303 size 72x72
      Appearance <- "DB_Field_Field{6,17}_HMI_Visualization"
   Rectangle "Rettangolo_118" at 1242,303 size 72x72
      Appearance <- "DB_Field_Field{6,18}_HMI_Visualization"
   Rectangle "Rettangolo_119" at 1314,303 size 72x72
      Appearance <- "DB_Field_Field{6,19}_HMI_Visualization"
   Rectangle "Rettangolo_120" at 1386,303 size 72x72
      Appearance <- "DB_Field_Field{6,20}_HMI_Visualization"
   Rectangle "Rettangolo_121" at 25,230 size 72x72
      Appearance <- "DB_Field_Field{7,1}_HMI_Visualization"
   Rectangle "Rettangolo_122" at 97,230 size 72x72
      Appearance <- "DB_Field_Field{7,2}_HMI_Visualization"
   Rectangle "Rettangolo_123" at 168,230 size 72x72
      Appearance <- "DB_Field_Field{7,3}_HMI_Visualization"
   Rectangle "Rettangolo_124" at 240,230 size 72x72
      Appearance <- "DB_Field_Field{7,4}_HMI_Visualization"
   Rectangle "Rettangolo_125" at 311,230 size 72x72
      Appearance <- "DB_Field_Field{7,5}_HMI_Visualization"
   Rectangle "Rettangolo_126" at 383,230 size 72x72
      Appearance <- "DB_Field_Field{7,6}_HMI_Visualization"
   Rectangle "Rettangolo_127" at 454,230 size 72x72
      Appearance <- "DB_Field_Field{7,7}_HMI_Visualization"
   Rectangle "Rettangolo_128" at 526,230 size 72x72
      Appearance <- "DB_Field_Field{7,8}_HMI_Visualization"
   Rectangle "Rettangolo_129" at 598,230 size 72x72
      Appearance <- "DB_Field_Field{7,9}_HMI_Visualization"
   Rectangle "Rettangolo_130" at 670,230 size 72x72
      Appearance <- "DB_Field_Field{7,10}_HMI_Visualization"
   Rectangle "Rettangolo_131" at 741,230 size 72x72
      Appearance <- "DB_Field_Field{7,11}_HMI_Visualization"
   Rectangle "Rettangolo_132" at 813,230 size 72x72
      Appearance <- "DB_Field_Field{7,12}_HMI_Visualization"
   Rectangle "Rettangolo_133" at 884,230 size 72x72
      Appearance <- "DB_Field_Field{7,13}_HMI_Visualization"
   Rectangle "Rettangolo_134" at 956,230 size 72x72
      Appearance <- "DB_Field_Field{7,14}_HMI_Visualization"
   Rectangle "Rettangolo_135" at 1027,230 size 72x72
      Appearance <- "DB_Field_Field{7,15}_HMI_Visualization"
   Rectangle "Rettangolo_136" at 1099,230 size 72x72
      Appearance <- "DB_Field_Field{7,16}_HMI_Visualization"
   Rectangle "Rettangolo_137" at 1170,230 size 72x72
      Appearance <- "DB_Field_Field{7,17}_HMI_Visualization"
   Rectangle "Rettangolo_138" at 1242,230 size 72x72
      Appearance <- "DB_Field_Field{7,18}_HMI_Visualization"
   Rectangle "Rettangolo_139" at 1314,230 size 72x72
      Appearance <- "DB_Field_Field{7,19}_HMI_Visualization"
   Rectangle "Rettangolo_140" at 1386,230 size 72x72
      Appearance <- "DB_Field_Field{7,20}_HMI_Visualization"
   Rectangle "Rettangolo_141" at 25,158 size 72x72
      Appearance <- "DB_Field_Field{8,1}_HMI_Visualization"
   Rectangle "Rettangolo_142" at 97,158 size 72x72
      Appearance <- "DB_Field_Field{8,2}_HMI_Visualization"
   Rectangle "Rettangolo_143" at 168,158 size 72x72
      Appearance <- "DB_Field_Field{8,3}_HMI_Visualization"
   Rectangle "Rettangolo_144" at 240,158 size 72x72
      Appearance <- "DB_Field_Field{8,4}_HMI_Visualization"
   Rectangle "Rettangolo_145" at 311,158 size 72x72
      Appearance <- "DB_Field_Field{8,5}_HMI_Visualization"
   Rectangle "Rettangolo_146" at 383,158 size 72x72
      Appearance <- "DB_Field_Field{8,6}_HMI_Visualization"
   Rectangle "Rettangolo_147" at 454,158 size 72x72
      Appearance <- "DB_Field_Field{8,7}_HMI_Visualization"
   Rectangle "Rettangolo_148" at 526,158 size 72x72
      Appearance <- "DB_Field_Field{8,8}_HMI_Visualization"
   Rectangle "Rettangolo_149" at 598,158 size 72x72
      Appearance <- "DB_Field_Field{8,9}_HMI_Visualization"
   Rectangle "Rettangolo_150" at 670,158 size 72x72
      Appearance <- "DB_Field_Field{8,10}_HMI_Visualization"
   Rectangle "Rettangolo_151" at 741,158 size 72x72
      Appearance <- "DB_Field_Field{8,11}_HMI_Visualization"
   Rectangle "Rettangolo_152" at 813,158 size 72x72
      Appearance <- "DB_Field_Field{8,12}_HMI_Visualization"
   Rectangle "Rettangolo_153" at 884,158 size 72x72
      Appearance <- "DB_Field_Field{8,13}_HMI_Visualization"
   Rectangle "Rettangolo_154" at 956,158 size 72x72
      Appearance <- "DB_Field_Field{8,14}_HMI_Visualization"
   Rectangle "Rettangolo_155" at 1027,158 size 72x72
      Appearance <- "DB_Field_Field{8,15}_HMI_Visualization"
   Rectangle "Rettangolo_156" at 1099,158 size 72x72
      Appearance <- "DB_Field_Field{8,16}_HMI_Visualization"
   Rectangle "Rettangolo_157" at 1170,158 size 72x72
      Appearance <- "DB_Field_Field{8,17}_HMI_Visualization"
   Rectangle "Rettangolo_158" at 1242,158 size 72x72
      Appearance <- "DB_Field_Field{8,18}_HMI_Visualization"
   Rectangle "Rettangolo_159" at 1314,158 size 72x72
      Appearance <- "DB_Field_Field{8,19}_HMI_Visualization"
   Rectangle "Rettangolo_160" at 1386,158 size 72x72
      Appearance <- "DB_Field_Field{8,20}_HMI_Visualization"
   Rectangle "Rettangolo_161" at 25,85 size 72x72
      Appearance <- "DB_Field_Field{9,1}_HMI_Visualization"
   Rectangle "Rettangolo_162" at 97,85 size 72x72
      Appearance <- "DB_Field_Field{9,2}_HMI_Visualization"
   Rectangle "Rettangolo_163" at 168,85 size 72x72
      Appearance <- "DB_Field_Field{9,3}_HMI_Visualization"
   Rectangle "Rettangolo_164" at 240,85 size 72x72
      Appearance <- "DB_Field_Field{9,4}_HMI_Visualization"
   Rectangle "Rettangolo_165" at 311,85 size 72x72
      Appearance <- "DB_Field_Field{9,5}_HMI_Visualization"
   Rectangle "Rettangolo_166" at 383,85 size 72x72
      Appearance <- "DB_Field_Field{9,6}_HMI_Visualization"
   Rectangle "Rettangolo_167" at 454,85 size 72x72
      Appearance <- "DB_Field_Field{9,7}_HMI_Visualization"
   Rectangle "Rettangolo_168" at 526,85 size 72x72
      Appearance <- "DB_Field_Field{9,8}_HMI_Visualization"
   Rectangle "Rettangolo_169" at 598,85 size 72x72
      Appearance <- "DB_Field_Field{9,9}_HMI_Visualization"
   Rectangle "Rettangolo_170" at 670,85 size 72x72
      Appearance <- "DB_Field_Field{9,10}_HMI_Visualization"
   Rectangle "Rettangolo_171" at 741,85 size 72x72
      Appearance <- "DB_Field_Field{9,11}_HMI_Visualization"
   Rectangle "Rettangolo_172" at 813,85 size 72x72
      Appearance <- "DB_Field_Field{9,12}_HMI_Visualization"
   Rectangle "Rettangolo_173" at 884,85 size 72x72
      Appearance <- "DB_Field_Field{9,13}_HMI_Visualization"
   Rectangle "Rettangolo_174" at 956,85 size 72x72
      Appearance <- "DB_Field_Field{9,14}_HMI_Visualization"
   Rectangle "Rettangolo_175" at 1027,85 size 72x72
      Appearance <- "DB_Field_Field{9,15}_HMI_Visualization"
   Rectangle "Rettangolo_176" at 1099,85 size 72x72
      Appearance <- "DB_Field_Field{9,16}_HMI_Visualization"
   Rectangle "Rettangolo_177" at 1170,85 size 72x72
      Appearance <- "DB_Field_Field{9,17}_HMI_Visualization"
   Rectangle "Rettangolo_178" at 1242,85 size 72x72
      Appearance <- "DB_Field_Field{9,18}_HMI_Visualization"
   Rectangle "Rettangolo_179" at 1314,85 size 72x72
      Appearance <- "DB_Field_Field{9,19}_HMI_Visualization"
   Rectangle "Rettangolo_180" at 1386,85 size 72x72
      Appearance <- "DB_Field_Field{9,20}_HMI_Visualization"
   Button "Pulsante_1" at 1480,476 size 216x91; TextOff 'LEFT'
      on Press: SetBit("DB_Commands_Cmd_SnakeLeft"); ResetBit("DB_Commands_Cmd_SnakeUp"); ResetBit("DB_Commands_Cmd_SnakeRight"); ResetBit("DB_Commands_Cmd_SnakeDown")
      ObjectEnable <- "DB_Commands_Sts_GameActive"
   Button "Pulsante_2" at 1696,476 size 216x91; TextOn 'RIGHT'; TextOff 'RIGHT'
      on Press: SetBit("DB_Commands_Cmd_SnakeRight"); ResetBit("DB_Commands_Cmd_SnakeUp"); ResetBit("DB_Commands_Cmd_SnakeLeft"); ResetBit("DB_Commands_Cmd_SnakeDown")
      ObjectEnable <- "DB_Commands_Sts_GameActive"
   Button "Pulsante_3" at 1588,384 size 216x91; TextOn 'UP'; TextOff 'UP'
      on Press: SetBit("DB_Commands_Cmd_SnakeUp"); ResetBit("DB_Commands_Cmd_SnakeDown"); ResetBit("DB_Commands_Cmd_SnakeLeft"); ResetBit("DB_Commands_Cmd_SnakeRight")
      ObjectEnable <- "DB_Commands_Sts_GameActive"
   Button "Pulsante_4" at 1589,568 size 216x91; TextOn 'DOWN'; TextOff 'DOWN'
      on Press: SetBit("DB_Commands_Cmd_SnakeDown"); ResetBit("DB_Commands_Cmd_SnakeUp"); ResetBit("DB_Commands_Cmd_SnakeLeft"); ResetBit("DB_Commands_Cmd_SnakeRight")
      ObjectEnable <- "DB_Commands_Sts_GameActive"
   IOField "Campo I/O_1" at 1573,82 size 246x77; FormatPattern 999999999
      ProcessValue <- "DB_Commands_Points_Actual"
   TextField "HmiScreenItemData_3" at 1598,16 size 196x54; Text 'POINTS'
   IOField "Campo I/O_2" at 1602,835 size 246x77; FormatPattern 999999999
      ProcessValue <- "DB_Commands_Points_BestGame"
   TextField "HmiScreenItemData_1" at 1627,769 size 196x54; Text 'BEST'
   Rectangle "Rettangolo_201" at 1211,792 size 253x112
      Appearance <- "DB_Commands_Cmd_Stop"
   Button "Pulsante_6" at 1212,792 size 253x112; TextOff 'TERMINA PARTITA'
      Appearance <- "DB_Commands_Cmd_Stop"
      on Press: SetBit("DB_Commands_Cmd_Stop")
   Rectangle "Rettangolo_202" at 923,792 size 253x112
      Appearance <- "DB_Commands_Sts_PauseActive"
   Button "Pulsante_5" at 923,793 size 253x112; TextOn 'PAUSA'; TextOff 'PAUSA'
      on Press: SetBit("DB_Commands_Cmd_Pause")
   Rectangle "Rettangolo_203" at 638,793 size 253x112
      Appearance <- "DB_Commands_Sts_GameActive"
   Button "Pulsante_7" at 639,794 size 253x112; TextOn 'START'; TextOff 'START'
      on Press: SetBit("DB_Commands_Cmd_Start")
   IOField "Campo I/O_3" at 27,832 size 246x77; FormatPattern 99.9; Unit  bloc/s
      ProcessValue <- "DB_Commands_Cmd_Speed"
   TextField "HmiScreenItemData_2" at 19,766 size 263x54; Text 'SPEED'
   Group "Group_1" at 25,85 size 1433x72
   Group "Group_2" at 25,158 size 1433x72
   Group "Group_3" at 25,230 size 1433x72
   Group "Group_4" at 25,303 size 1433x72
   Group "Group_5" at 25,375 size 1433x72
   Group "Group_6" at 25,448 size 1433x72
   Group "Group_7" at 25,520 size 1433x72
   Group "Group_8" at 25,593 size 1433x72
   Group "Group_9" at 25,665 size 1433x72
   Group "Group" at 25,13 size 1433x72
   IOField "Campo I/O_4" at 1573,235 size 246x77; FormatPattern 999999999
      ProcessValue <- "DB_Commands_Sts_SnakeLength"
   TextField "HmiScreenItemData_4" at 1598,169 size 196x54; Text 'LENGTH'
   Rectangle "Rettangolo_181" at 25,13 size 72x72
      Appearance <- "DB_Field_Field{10,1}_HMI_Visualization"
   Rectangle "Rettangolo_182" at 97,13 size 72x72
      Appearance <- "DB_Field_Field{10,2}_HMI_Visualization"
   Rectangle "Rettangolo_183" at 168,13 size 72x72
      Appearance <- "DB_Field_Field{10,3}_HMI_Visualization"
   Rectangle "Rettangolo_184" at 240,13 size 72x72
      Appearance <- "DB_Field_Field{10,4}_HMI_Visualization"
   Rectangle "Rettangolo_185" at 311,13 size 72x72
      Appearance <- "DB_Field_Field{10,5}_HMI_Visualization"
   Rectangle "Rettangolo_186" at 383,13 size 72x72
      Appearance <- "DB_Field_Field{10,6}_HMI_Visualization"
   Rectangle "Rettangolo_187" at 454,13 size 72x72
      Appearance <- "DB_Field_Field{10,7}_HMI_Visualization"
   Rectangle "Rettangolo_188" at 526,13 size 72x72
      Appearance <- "DB_Field_Field{10,8}_HMI_Visualization"
   Rectangle "Rettangolo_189" at 598,13 size 72x72
      Appearance <- "DB_Field_Field{10,9}_HMI_Visualization"
   Rectangle "Rettangolo_190" at 670,13 size 72x72
      Appearance <- "DB_Field_Field{10,10}_HMI_Visualization"
   Rectangle "Rettangolo_191" at 741,13 size 72x72
      Appearance <- "DB_Field_Field{10,11}_HMI_Visualization"
   Rectangle "Rettangolo_192" at 813,13 size 72x72
      Appearance <- "DB_Field_Field{10,12}_HMI_Visualization"
   Rectangle "Rettangolo_193" at 884,13 size 72x72
      Appearance <- "DB_Field_Field{10,13}_HMI_Visualization"
   Rectangle "Rettangolo_194" at 956,13 size 72x72
      Appearance <- "DB_Field_Field{10,14}_HMI_Visualization"
   Rectangle "Rettangolo_195" at 1027,13 size 72x72
      Appearance <- "DB_Field_Field{10,15}_HMI_Visualization"
   Rectangle "Rettangolo_196" at 1099,13 size 72x72
      Appearance <- "DB_Field_Field{10,16}_HMI_Visualization"
   Rectangle "Rettangolo_197" at 1170,13 size 72x72
      Appearance <- "DB_Field_Field{10,17}_HMI_Visualization"
   Rectangle "Rettangolo_198" at 1242,13 size 72x72
      Appearance <- "DB_Field_Field{10,18}_HMI_Visualization"
   Rectangle "Rettangolo_199" at 1314,13 size 72x72
      Appearance <- "DB_Field_Field{10,19}_HMI_Visualization"
   Rectangle "Rettangolo_200" at 1386,13 size 72x72
      Appearance <- "DB_Field_Field{10,20}_HMI_Visualization"

Template "Modello_1" 1920x1020
   Button "Template_Button" at 1840,960 size 78x58; TextOff 'Text'
   Button "Template_Button_1" at 1760,960 size 78x58; TextOff 'Text'
   Button "Template_Button_2" at 1680,960 size 78x58; TextOff 'Text'
   Button "Template_Button_3" at 1600,960 size 78x58; TextOff 'Text'
   Button "Template_Button_4" at 1520,960 size 78x58; TextOff 'Text'
   Button "Template_Button_5" at 1440,960 size 78x58; TextOff 'Text'
   Button "Template_Button_6" at 1360,960 size 78x58; TextOff 'Text'
   Button "Template_Button_7" at 1280,960 size 78x58; TextOff 'Text'
   Button "Template_Button_8" at 1200,960 size 78x58; TextOff 'Text'
   Button "Template_Button_9" at 1120,960 size 78x58; TextOff 'Text'
   Button "Template_Button_10" at 1040,960 size 78x58; TextOff 'Text'
   Button "Template_Button_11" at 960,960 size 78x58; TextOff 'Text'
   Button "Template_Button_12" at 881,960 size 78x58; TextOff 'Text'
   Button "Template_Button_13" at 801,960 size 78x58; TextOff 'Text'
   Button "Template_Button_14" at 721,960 size 78x58; TextOff 'Text'
   Button "Template_Button_15" at 641,960 size 78x58; TextOff 'Text'
   Button "Template_Button_16" at 561,960 size 78x58; TextOff 'Text'
   Button "Template_Button_17" at 481,960 size 78x58; TextOff 'Text'
   Button "Template_Button_18" at 401,960 size 78x58; TextOff 'Text'
   Button "Template_Button_19" at 321,960 size 78x58; TextOff 'Text'
   Button "Template_Button_20" at 241,960 size 78x58; TextOff 'Text'
   Button "Template_Button_21" at 161,960 size 78x58; TextOff 'Text'
   Button "Template_Button_22" at 81,960 size 78x58; TextOff 'Text'
   Button "Template_Button_23" at 1,960 size 78x58; TextOff 'Text'
*)